KUKA KRL program: EPS_2_26115_SA7002_A_20260219035537.src

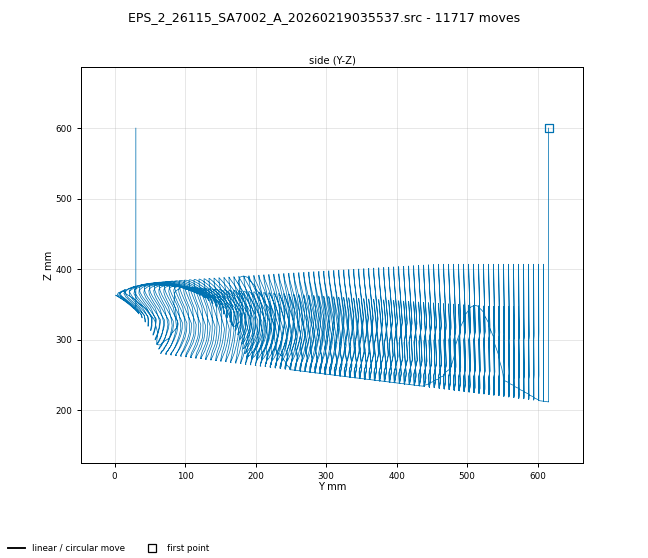
[picture p0: tool path of EPS_2_26115_SA7002_A_20260219035537.src, 11717 of 11719 moves have a stored position in this frame; points joined in program order, loops and branches not executed]
&ACCESS RVP
&REL 4
&COMMENT QRS 19112012
&PARAM EDITMASK = *
DEF PART()
EXT BAS (BAS_COMMAND :IN,REAL :IN )
INT I
BAS (#INITMOV,0 )

;KUKA QRS Post kuka4.cps  Date:22-06-2017 !

File_ID=3057

QRS_PRE_INIT()

;Init var - Until changes are made in qrs_pre_init
Outlet_Square_prg=0
Inlet_1_Square_prg=0
Inlet_2_Square_prg=0
Inlet_3_Square_prg=0
Inlet_4_Square_prg=0
Inlet_5_Square_prg=0

Outlet_1={X 0.000, Y 460.000, Z 306.500, B 0.000, E1 0.000 }
Inlet_1={X 0.000, Y 536.220, Z 246.500, B 0.000, E1 137.000 }
Outlet_1_type=201
Inlet_1_type=201
;QRS#1=Sidecore dimensions
;QRS#2=200-8" PVC SDR 35 Cut Back
;QRS#3=200-8" PVC SDR 35
;QRS#4=
;QRS#5=
;QRS#6=
;QRS#7=
;QRS#8=
;QRS#9=12-08 PSX
;QRS#10=12-08 PSX
;QRS#11=
;QRS#12=
;QRS#13=
;QRS#14=
;QRS#15=
;QRS#16=1220x127x686 2,25'
;QRS#17=EPS Height
;QRS#18=407
;QRS#19=*
;QRS#20= UPDATED VERSION 22-06-2017
;QRS#21=*
Outlet_Square=0100
Inlet_1_Square=0100
Inlet_2_Square=0
Inlet_3_Square=0
Inlet_4_Square=0
Inlet_5_Square=0
Mill_Square=1
Outlet_Square_Prg=214
Inlet_1_Square_prg=204

QRS_INIT()

$ADVANCE=5

; T1
PTP {E1 173.6,E2 173.6}
PTP {X 0,Y 615.51,A -85,B 0,C 180,E1 173.6,E2 173.6,E3 0,E4 0,E5 0,E6 0}
QRS_SPEED_INIT()
LIN {X 0,Y 615.51,Z 600,A -85,B 0,C 180,E1 173.6,E2 173.6,E3 0,E4 0,E5 0,E6 0} C_VEL
LIN {X 0,Y 615.51,Z 221.874,A -85,B 0,C 180,E1 173.6,E2 173.6} C_VEL
LIN {X 0,Y 615.51,Z 213.701,A -85,B 0,C 180,E1 173.6,E2 173.6} C_VEL
LIN {X 0,Y 615.491,Z 211.701,A -85,B 0,C 180,E1 173.414,E2 173.414} C_VEL
LIN {X 0,Y 615.474,Z 211.7,A -85,B 0,C 180,E1 170.802,E2 170.802} C_VEL
LIN {X 0,Y 615.475,Z 211.7,A -85,B 0,C 180,E1 168.808,E2 168.808} C_VEL
LIN {X 0,Y 615.494,Z 211.996,A -85,B 0,C 180,E1 168.141,E2 168.141} C_VEL
LIN {X 0,Y 615.484,Z 215.315,A -85,B 0,C 180,E1 165.452,E2 165.452} C_VEL
LIN {X 0,Y 615.469,Z 218.575,A -85,B 0,C 180,E1 162.73,E2 162.73} C_VEL
LIN {X 0,Y 615.439,Z 221.126,A -85,B 0,C 180,E1 160.662,E2 160.662} C_VEL
LIN {X 0,Y 615.437,Z 223.859,A -85,B 0,C 180,E1 158.568,E2 158.568} C_VEL
LIN {X 0,Y 615.482,Z 227.285,A -85,B 0,C 180,E1 155.991,E2 155.991} C_VEL
LIN {X 0,Y 615.455,Z 230.578,A -85,B 0,C 180,E1 153.556,E2 153.556} C_VEL
LIN {X 0,Y 615.427,Z 233.628,A -85,B 0,C 180,E1 151.341,E2 151.341} C_VEL
LIN {X 0,Y 615.423,Z 237.001,A -85,B 0,C 180,E1 148.923,E2 148.923} C_VEL
LIN {X 0,Y 615.475,Z 240.459,A -85,B 0,C 180,E1 146.467,E2 146.467} C_VEL
LIN {X 0,Y 615.481,Z 243.27,A -85,B 0,C 180,E1 144.536,E2 144.536} C_VEL
LIN {X 0,Y 615.498,Z 256.266,A -85,B 0,C 180,E1 144.248,E2 144.248} C_VEL
LIN {X 0,Y 615.471,Z 267.884,A -85,B 0,C 180,E1 143.87,E2 143.87} C_VEL
LIN {X 0,Y 615.442,Z 279.091,A -85,B 0,C 180,E1 143.384,E2 143.384} C_VEL
LIN {X 0,Y 615.469,Z 290.355,A -85,B 0,C 180,E1 142.759,E2 142.759} C_VEL
LIN {X 0,Y 615.495,Z 301.31,A -85,B 0,C 180,E1 141.986,E2 141.986} C_VEL
LIN {X 0,Y 615.498,Z 311.464,A -85,B 0,C 180,E1 141.099,E2 141.099} C_VEL
LIN {X 0,Y 615.494,Z 320.701,A -85,B 0,C 180,E1 140.081,E2 140.081} C_VEL
LIN {X 0,Y 615.496,Z 327.529,A -85,B 0,C 180,E1 139.151,E2 139.151} C_VEL
LIN {X 0,Y 615.496,Z 333.051,A -85,B 0,C 180,E1 138.224,E2 138.224} C_VEL
LIN {X 0,Y 615.495,Z 337.464,A -85,B 0,C 180,E1 137.301,E2 137.301} C_VEL
LIN {X 0,Y 615.497,Z 340.908,A -85,B 0,C 180,E1 136.381,E2 136.381} C_VEL
LIN {X 0,Y 615.498,Z 344.341,A -85,B 0,C 180,E1 135.067,E2 135.067} C_VEL
LIN {X 0,Y 615.495,Z 345.888,A -85,B 0,C 180,E1 134.001,E2 134.001} C_VEL
LIN {X 0,Y 615.496,Z 346.371,A -85,B 0,C 180,E1 133.051,E2 133.051} C_VEL
LIN {X 0,Y 615.498,Z 346.02,A -85,B 0,C 180,E1 132.084,E2 132.084} C_VEL
LIN {X 0,Y 615.495,Z 344.785,A -85,B 0,C 180,E1 131.098,E2 131.098} C_VEL
LIN {X 0,Y 615.493,Z 341.613,A -85,B 0,C 180,E1 129.749,E2 129.749} C_VEL
LIN {X 0,Y 615.492,Z 336.93,A -85,B 0,C 180,E1 128.484,E2 128.484} C_VEL
LIN {X 0,Y 615.497,Z 331.67,A -85,B 0,C 180,E1 127.434,E2 127.434} C_VEL
LIN {X 0,Y 615.496,Z 325.251,A -85,B 0,C 180,E1 126.424,E2 126.424} C_VEL
LIN {X 0,Y 615.493,Z 317.173,A -85,B 0,C 180,E1 125.414,E2 125.414} C_VEL
LIN {X 0,Y 615.497,Z 308.507,A -85,B 0,C 180,E1 124.533,E2 124.533} C_VEL
LIN {X 0,Y 615.498,Z 299.472,A -85,B 0,C 180,E1 123.78,E2 123.78} C_VEL
LIN {X 0,Y 615.481,Z 288.508,A -85,B 0,C 180,E1 123.041,E2 123.041} C_VEL
LIN {X 0,Y 615.495,Z 276.332,A -85,B 0,C 180,E1 122.395,E2 122.395} C_VEL
LIN {X 0,Y 615.48,Z 263.674,A -85,B 0,C 180,E1 121.888,E2 121.888} C_VEL
LIN {X 0,Y 615.494,Z 251.238,A -85,B 0,C 180,E1 121.535,E2 121.535} C_VEL
LIN {X 0,Y 615.485,Z 243.192,A -85,B 0,C 180,E1 121.367,E2 121.367} C_VEL
LIN {X 0,Y 615.492,Z 239.045,A -85,B 0,C 180,E1 118.455,E2 118.455} C_VEL
LIN {X 0,Y 615.476,Z 235.021,A -85,B 0,C 180,E1 115.571,E2 115.571} C_VEL
LIN {X 0,Y 615.475,Z 231.242,A -85,B 0,C 180,E1 112.844,E2 112.844} C_VEL
LIN {X 0,Y 615.485,Z 227.434,A -85,B 0,C 180,E1 110.032,E2 110.032} C_VEL
LIN {X 0,Y 615.465,Z 224.676,A -85,B 0,C 180,E1 107.957,E2 107.957} C_VEL
LIN {X 0,Y 615.45,Z 221.985,A -85,B 0,C 180,E1 105.906,E2 105.906} C_VEL
LIN {X 0,Y 615.439,Z 219.39,A -85,B 0,C 180,E1 103.875,E2 103.875} C_VEL
LIN {X 0,Y 615.481,Z 216.126,A -85,B 0,C 180,E1 101.193,E2 101.193} C_VEL
LIN {X 0,Y 615.476,Z 212.873,A -85,B 0,C 180,E1 98.536,E2 98.536} C_VEL
LIN {X 0,Y 615.485,Z 212.061,A -85,B 0,C 180,E1 97.875,E2 97.875} C_VEL
LIN {X 0,Y 615.497,Z 211.7,A -85,B 0,C 180,E1 96.556,E2 96.556} C_VEL
LIN {X 0,Y 615.482,Z 211.7,A -85,B 0,C 180,E1 93.928,E2 93.928} C_VEL
LIN {X 0,Y 615.487,Z 211.696,A -85,B 0,C 180,E1 91.308,E2 91.308} C_VEL
LIN {X 0,Y 615.484,Z 211.696,A -85,B 0,C 180,E1 88.691,E2 88.691} C_VEL
LIN {X 0,Y 615.476,Z 211.7,A -85,B 0,C 180,E1 86.071,E2 86.071} C_VEL
LIN {X 0,Y 615.491,Z 211.702,A -85,B 0,C 180,E1 83.402,E2 83.402} C_VEL
LIN {X 0,Y 615.475,Z 211.701,A -85,B 0,C 180,E1 80.801,E2 80.801} C_VEL
LIN {X 0,Y 615.468,Z 211.7,A -85,B 0,C 180,E1 78.139,E2 78.139} C_VEL
LIN {X 0,Y 615.482,Z 211.697,A -85,B 0,C 180,E1 75.451,E2 75.451} C_VEL
LIN {X 0,Y 615.497,Z 211.699,A -85,B 0,C 180,E1 72.729,E2 72.729} C_VEL
LIN {X 0,Y 615.481,Z 211.698,A -85,B 0,C 180,E1 69.967,E2 69.967} C_VEL
LIN {X 0,Y 615.49,Z 211.695,A -85,B 0,C 180,E1 67.155,E2 67.155} C_VEL
LIN {X 0,Y 615.496,Z 211.7,A -85,B 0,C 180,E1 64.284,E2 64.284} C_VEL
LIN {X 0,Y 615.489,Z 211.695,A -85,B 0,C 180,E1 61.342,E2 61.342} C_VEL
LIN {X 0,Y 615.47,Z 211.699,A -85,B 0,C 180,E1 58.913,E2 58.913} C_VEL
LIN {X 0,Y 615.466,Z 211.7,A -85,B 0,C 180,E1 56.466,E2 56.466} C_VEL
LIN {X 0,Y 615.465,Z 211.7,A -85,B 0,C 180,E1 54.166,E2 54.166} C_VEL
LIN {X 0,Y 615.487,Z 211.696,A -85,B 0,C 180,E1 51.931,E2 51.931} C_VEL
LIN {X 0,Y 615.486,Z 211.696,A -85,B 0,C 180,E1 49.393,E2 49.393} C_VEL
LIN {X 0,Y 615.475,Z 211.7,A -85,B 0,C 180,E1 46.754,E2 46.754} C_VEL
LIN {X 0,Y 615.495,Z 211.699,A -85,B 0,C 180,E1 43.998,E2 43.998} C_VEL
LIN {X 0,Y 615.466,Z 211.7,A -85,B 0,C 180,E1 41.092,E2 41.092} C_VEL
LIN {X 0,Y 615.468,Z 211.701,A -85,B 0,C 180,E1 38.904,E2 38.904} C_VEL
LIN {X 0,Y 615.476,Z 211.698,A -85,B 0,C 180,E1 36.424,E2 36.424} C_VEL
LIN {X 0,Y 615.493,Z 211.698,A -85,B 0,C 180,E1 33.535,E2 33.535} C_VEL
LIN {X 0,Y 615.488,Z 211.702,A -85,B 0,C 180,E1 30.918,E2 30.918} C_VEL
LIN {X 0,Y 615.492,Z 211.699,A -85,B 0,C 180,E1 28.451,E2 28.451} C_VEL
LIN {X 0,Y 615.474,Z 211.698,A -85,B 0,C 180,E1 25.566,E2 25.566} C_VEL
LIN {X 0,Y 615.478,Z 211.701,A -85,B 0,C 180,E1 22.843,E2 22.843} C_VEL
LIN {X 0,Y 615.474,Z 211.7,A -85,B 0,C 180,E1 20.553,E2 20.553} C_VEL
LIN {X 0,Y 615.497,Z 211.698,A -85,B 0,C 180,E1 17.955,E2 17.955} C_VEL
LIN {X 0,Y 615.478,Z 211.7,A -85,B 0,C 180,E1 15.225,E2 15.225} C_VEL
LIN {X 0,Y 615.488,Z 211.695,A -85,B 0,C 180,E1 12.529,E2 12.529} C_VEL
LIN {X 0,Y 615.483,Z 211.698,A -85,B 0,C 180,E1 9.861,E2 9.861} C_VEL
LIN {X 0,Y 615.486,Z 211.701,A -85,B 0,C 180,E1 7.214,E2 7.214} C_VEL
LIN {X 0,Y 615.496,Z 211.697,A -85,B 0,C 180,E1 4.583,E2 4.583} C_VEL
LIN {X 0,Y 615.471,Z 211.7,A -85,B 0,C 180,E1 1.962,E2 1.962} C_VEL
LIN {X 0,Y 615.467,Z 211.7,A -85,B 0,C 180,E1 -0.655,E2 -0.655} C_VEL
LIN {X 0,Y 615.484,Z 211.698,A -85,B 0,C 180,E1 -3.274,E2 -3.274} C_VEL
LIN {X 0,Y 615.495,Z 211.699,A -85,B 0,C 180,E1 -5.899,E2 -5.899} C_VEL
LIN {X 0,Y 615.485,Z 211.7,A -85,B 0,C 180,E1 -8.538,E2 -8.538} C_VEL
LIN {X 0,Y 615.49,Z 211.695,A -85,B 0,C 180,E1 -11.194,E2 -11.194} C_VEL
LIN {X 0,Y 615.475,Z 211.699,A -85,B 0,C 180,E1 -13.927,E2 -13.927} C_VEL
LIN {X 0,Y 615.488,Z 211.7,A -85,B 0,C 180,E1 -16.587,E2 -16.587} C_VEL
LIN {X 0,Y 615.486,Z 211.698,A -85,B 0,C 180,E1 -19.339,E2 -19.339} C_VEL
LIN {X 0,Y 615.466,Z 211.7,A -85,B 0,C 180,E1 -22.138,E2 -22.138} C_VEL
LIN {X 0,Y 615.493,Z 211.7,A -85,B 0,C 180,E1 -24.992,E2 -24.992} C_VEL
LIN {X 0,Y 615.497,Z 211.696,A -85,B 0,C 180,E1 -27.178,E2 -27.178} C_VEL
LIN {X 0,Y 615.499,Z 211.7,A -85,B 0,C 180,E1 -29.796,E2 -29.796} C_VEL
LIN {X 0,Y 615.488,Z 211.698,A -85,B 0,C 180,E1 -32.458,E2 -32.458} C_VEL
LIN {X 0,Y 615.497,Z 211.696,A -85,B 0,C 180,E1 -34.815,E2 -34.815} C_VEL
LIN {X 0,Y 615.476,Z 211.7,A -85,B 0,C 180,E1 -37.244,E2 -37.244} C_VEL
LIN {X 0,Y 615.469,Z 211.7,A -85,B 0,C 180,E1 -39.752,E2 -39.752} C_VEL
LIN {X 0,Y 615.473,Z 211.699,A -85,B 0,C 180,E1 -42.355,E2 -42.355} C_VEL
LIN {X 0,Y 615.49,Z 211.698,A -85,B 0,C 180,E1 -45.069,E2 -45.069} C_VEL
LIN {X 0,Y 615.484,Z 211.699,A -85,B 0,C 180,E1 -47.921,E2 -47.921} C_VEL
LIN {X 0,Y 615.491,Z 211.696,A -85,B 0,C 180,E1 -50.938,E2 -50.938} C_VEL
LIN {X 0,Y 615.486,Z 211.701,A -85,B 0,C 180,E1 -53.575,E2 -53.575} C_VEL
LIN {X 0,Y 615.49,Z 211.816,A -85,B 0,C 180,E1 -54.535,E2 -54.535} C_VEL
LIN {X 0,Y 615.437,Z 220.579,A -85,B 0,C 180,E1 -57.151,E2 -57.151} C_VEL
LIN {X 0,Y 615.425,Z 228.512,A -85,B 0,C 180,E1 -59.457,E2 -59.457} C_VEL
LIN {X 0,Y 615.48,Z 237.754,A -85,B 0,C 180,E1 -62.084,E2 -62.084} C_VEL
LIN {X 0,Y 615.47,Z 247.263,A -85,B 0,C 180,E1 -64.718,E2 -64.718} C_VEL
LIN {X 0,Y 615.465,Z 256.236,A -85,B 0,C 180,E1 -67.154,E2 -67.154} C_VEL
LIN {X 0,Y 615.483,Z 266.781,A -85,B 0,C 180,E1 -69.967,E2 -69.967} C_VEL
LIN {X 0,Y 615.484,Z 277.325,A -85,B 0,C 180,E1 -72.729,E2 -72.729} C_VEL
LIN {X 0,Y 615.464,Z 287.861,A -85,B 0,C 180,E1 -75.45,E2 -75.45} C_VEL
LIN {X 0,Y 615.484,Z 298.39,A -85,B 0,C 180,E1 -78.139,E2 -78.139} C_VEL
LIN {X 0,Y 615.496,Z 299.207,A -85,B 0,C 180,E1 -78.348,E2 -78.348} C_VEL
LIN {X 0,Y 615.497,Z 313.809,A -85,B 0,C 180,E1 -78.64,E2 -78.64} C_VEL
LIN {X 0,Y 615.455,Z 326.946,A -85,B 0,C 180,E1 -79.05,E2 -79.05} C_VEL
LIN {X 0,Y 615.447,Z 338.766,A -85,B 0,C 180,E1 -79.555,E2 -79.555} C_VEL
LIN {X 0,Y 615.497,Z 349.381,A -85,B 0,C 180,E1 -80.138,E2 -80.138} C_VEL
LIN {X 0,Y 615.498,Z 360.228,A -85,B 0,C 180,E1 -80.884,E2 -80.884} C_VEL
LIN {X 0,Y 615.497,Z 370.808,A -85,B 0,C 180,E1 -81.794,E2 -81.794} C_VEL
LIN {X 0,Y 615.498,Z 378.603,A -85,B 0,C 180,E1 -82.619,E2 -82.619} C_VEL
LIN {X 0,Y 615.496,Z 386.201,A -85,B 0,C 180,E1 -83.608,E2 -83.608} C_VEL
LIN {X 0,Y 615.498,Z 393.203,A -85,B 0,C 180,E1 -84.759,E2 -84.759} C_VEL
LIN {X 0,Y 615.494,Z 397.85,A -85,B 0,C 180,E1 -85.743,E2 -85.743} C_VEL
LIN {X 0,Y 615.494,Z 401.398,A -85,B 0,C 180,E1 -86.727,E2 -86.727} C_VEL
LIN {X 0,Y 615.497,Z 403.232,A -85,B 0,C 180,E1 -87.382,E2 -87.382} C_VEL
LIN {X 0,Y 615.5,Z 404.607,A -85,B 0,C 180,E1 -88.037,E2 -88.037} C_VEL
LIN {X 0,Y 615.496,Z 406.173,A -85,B 0,C 180,E1 -89.345,E2 -89.345} C_VEL
LIN {X 0,Y 615.494,Z 406.389,A -85,B 0,C 180,E1 -90,E2 -90} C_VEL
LIN {X 0,Y 615.495,Z 405.58,A -85,B 0,C 180,E1 -91.308,E2 -91.308} C_VEL
LIN {X 0,Y 615.5,Z 404.608,A -85,B 0,C 180,E1 -91.963,E2 -91.963} C_VEL
LIN {X 0,Y 615.497,Z 403.234,A -85,B 0,C 180,E1 -92.617,E2 -92.617} C_VEL
LIN {X 0,Y 615.496,Z 400.351,A -85,B 0,C 180,E1 -93.6,E2 -93.6} C_VEL
LIN {X 0,Y 615.498,Z 396.443,A -85,B 0,C 180,E1 -94.584,E2 -94.584} C_VEL
LIN {X 0,Y 615.499,Z 391.407,A -85,B 0,C 180,E1 -95.569,E2 -95.569} C_VEL
LIN {X 0,Y 615.497,Z 384.871,A -85,B 0,C 180,E1 -96.583,E2 -96.583} C_VEL
LIN {X 0,Y 615.497,Z 377.137,A -85,B 0,C 180,E1 -97.545,E2 -97.545} C_VEL
LIN {X 0,Y 615.498,Z 369.049,A -85,B 0,C 180,E1 -98.371,E2 -98.371} C_VEL
LIN {X 0,Y 615.499,Z 359.173,A -85,B 0,C 180,E1 -99.198,E2 -99.198} C_VEL
LIN {X 0,Y 615.486,Z 347.989,A -85,B 0,C 180,E1 -99.945,E2 -99.945} C_VEL
LIN {X 0,Y 615.445,Z 337.038,A -85,B 0,C 180,E1 -100.527,E2 -100.527} C_VEL
LIN {X 0,Y 615.461,Z 324.766,A -85,B 0,C 180,E1 -101.031,E2 -101.031} C_VEL
LIN {X 0,Y 615.499,Z 312.081,A -85,B 0,C 180,E1 -101.401,E2 -101.401} C_VEL
LIN {X 0,Y 615.496,Z 299.21,A -85,B 0,C 180,E1 -101.651,E2 -101.651} C_VEL
LIN {X 0,Y 615.465,Z 289.075,A -85,B 0,C 180,E1 -104.24,E2 -104.24} C_VEL
LIN {X 0,Y 615.49,Z 278.641,A -85,B 0,C 180,E1 -106.928,E2 -106.928} C_VEL
LIN {X 0,Y 615.487,Z 268.106,A -85,B 0,C 180,E1 -109.685,E2 -109.685} C_VEL
LIN {X 0,Y 615.491,Z 258.087,A -85,B 0,C 180,E1 -112.346,E2 -112.346} C_VEL
LIN {X 0,Y 615.456,Z 248.325,A -85,B 0,C 180,E1 -114.993,E2 -114.993} C_VEL
LIN {X 0,Y 615.494,Z 239.076,A -85,B 0,C 180,E1 -117.545,E2 -117.545} C_VEL
LIN {X 0,Y 615.44,Z 229.836,A -85,B 0,C 180,E1 -120.162,E2 -120.162} C_VEL
LIN {X 0,Y 615.421,Z 221.905,A -85,B 0,C 180,E1 -122.461,E2 -122.461} C_VEL
LIN {X 0,Y 615.454,Z 213.969,A -85,B 0,C 180,E1 -124.817,E2 -124.817} C_VEL
LIN {X 0,Y 615.492,Z 211.697,A -85,B 0,C 180,E1 -125.514,E2 -125.514} C_VEL
LIN {X 0,Y 615.486,Z 211.699,A -85,B 0,C 180,E1 -128.068,E2 -128.068} C_VEL
LIN {X 0,Y 615.484,Z 211.7,A -85,B 0,C 180,E1 -130.606,E2 -130.606} C_VEL
LIN {X 0,Y 615.497,Z 211.697,A -85,B 0,C 180,E1 -133.243,E2 -133.243} C_VEL
LIN {X 0,Y 615.474,Z 211.7,A -85,B 0,C 180,E1 -136.003,E2 -136.003} C_VEL
LIN {X 0,Y 615.487,Z 211.7,A -85,B 0,C 180,E1 -138.525,E2 -138.525} C_VEL
LIN {X 0,Y 615.495,Z 211.696,A -85,B 0,C 180,E1 -141.096,E2 -141.096} C_VEL
LIN {X 0,Y 615.487,Z 211.698,A -85,B 0,C 180,E1 -143.574,E2 -143.574} C_VEL
LIN {X 0,Y 615.495,Z 211.701,A -85,B 0,C 180,E1 -145.978,E2 -145.978} C_VEL
LIN {X 0,Y 615.484,Z 211.7,A -85,B 0,C 180,E1 -148.913,E2 -148.913} C_VEL
LIN {X 0,Y 615.475,Z 211.7,A -85,B 0,C 180,E1 -151.551,E2 -151.551} C_VEL
LIN {X 0,Y 615.498,Z 211.7,A -85,B 0,C 180,E1 -154.284,E2 -154.284} C_VEL
LIN {X 0,Y 615.493,Z 211.697,A -85,B 0,C 180,E1 -157.155,E2 -157.155} C_VEL
LIN {X 0,Y 615.475,Z 211.7,A -85,B 0,C 180,E1 -159.966,E2 -159.966} C_VEL
LIN {X 0,Y 615.497,Z 211.699,A -85,B 0,C 180,E1 -162.729,E2 -162.729} C_VEL
LIN {X 0,Y 615.481,Z 211.7,A -85,B 0,C 180,E1 -165.45,E2 -165.45} C_VEL
LIN {X 0,Y 615.484,Z 211.699,A -85,B 0,C 180,E1 -168.138,E2 -168.138} C_VEL
LIN {X 0,Y 615.496,Z 211.698,A -85,B 0,C 180,E1 -170.8,E2 -170.8} C_VEL
LIN {X 0,Y 615.474,Z 211.7,A -85,B 0,C 180,E1 -173.442,E2 -173.442} C_VEL
LIN {X 0,Y 615.488,Z 211.701,A -85,B 0,C 180,E1 -176.07,E2 -176.07} C_VEL
LIN {X 0,Y 615.491,Z 211.696,A -85,B 0,C 180,E1 -178.69,E2 -178.69} C_VEL
LIN {X 0,Y 615.496,Z 211.7,A -85,B 0,C 180,E1 -181.307,E2 -181.307} C_VEL
LIN {X 0,Y 615.477,Z 211.7,A -85,B 0,C 180,E1 -183.927,E2 -183.927} C_VEL
LIN {X 0,Y 615.491,Z 211.701,A -85,B 0,C 180,E1 -186.586,E2 -186.586} C_VEL
LIN {X 0,Y 614.803,Z 211.847,A -85,B 0,C 180,E1 -187.132,E2 -187.132} C_VEL
LIN {X 0,Y 611.958,Z 212.259,A -85,B 0,C 180,E1 -188.018,E2 -188.018} C_VEL
LIN {X 0,Y 609.568,Z 212.568,A -85,B 0,C 180,E1 -188.731,E2 -188.731} C_VEL
LIN {X 0,Y 608.539,Z 212.686,A -85,B 0,C 180,E1 -189.28,E2 -189.28} C_VEL
LIN {X 0,Y 608.454,Z 212.695,A -85,B 0,C 180,E1 -189.466,E2 -189.466} C_VEL
LIN {X 0,Y 608.44,Z 212.697,A -85,B 0,C 180,E1 -191.323,E2 -191.323} C_VEL
LIN {X 0,Y 608.449,Z 213.027,A -85,B 0,C 180,E1 -191.999,E2 -191.999} C_VEL
LIN {X 0,Y 608.442,Z 216.384,A -85,B 0,C 180,E1 -194.72,E2 -194.72} C_VEL
LIN {X 0,Y 608.437,Z 219.656,A -85,B 0,C 180,E1 -197.476,E2 -197.476} C_VEL
LIN {X 0,Y 608.426,Z 223.103,A -85,B 0,C 180,E1 -200.274,E2 -200.274} C_VEL
LIN {X 0,Y 608.374,Z 226.848,A -85,B 0,C 180,E1 -203.125,E2 -203.125} C_VEL
LIN {X 0,Y 608.389,Z 230.305,A -85,B 0,C 180,E1 -205.706,E2 -205.706} C_VEL
LIN {X 0,Y 608.366,Z 234.261,A -85,B 0,C 180,E1 -208.603,E2 -208.603} C_VEL
LIN {X 0,Y 608.396,Z 236.953,A -85,B 0,C 180,E1 -210.547,E2 -210.547} C_VEL
LIN {X 0,Y 608.388,Z 240.222,A -85,B 0,C 180,E1 -212.882,E2 -212.882} C_VEL
LIN {X 0,Y 608.407,Z 243.684,A -85,B 0,C 180,E1 -215.329,E2 -215.329} C_VEL
LIN {X 0,Y 608.536,Z 257.877,A -85,B 0,C 180,E1 -215.663,E2 -215.663} C_VEL
LIN {X 0,Y 608.509,Z 270.159,A -85,B 0,C 180,E1 -216.086,E2 -216.086} C_VEL
LIN {X 0,Y 608.464,Z 281.367,A -85,B 0,C 180,E1 -216.603,E2 -216.603} C_VEL
LIN {X 0,Y 608.475,Z 292.485,A -85,B 0,C 180,E1 -217.255,E2 -217.255} C_VEL
LIN {X 0,Y 608.483,Z 302.616,A -85,B 0,C 180,E1 -217.993,E2 -217.993} C_VEL
LIN {X 0,Y 608.459,Z 311.688,A -85,B 0,C 180,E1 -218.799,E2 -218.799} C_VEL
LIN {X 0,Y 608.467,Z 319.57,A -85,B 0,C 180,E1 -219.652,E2 -219.652} C_VEL
LIN {X 0,Y 608.451,Z 327.678,A -85,B 0,C 180,E1 -220.736,E2 -220.736} C_VEL
LIN {X 0,Y 608.444,Z 334.345,A -85,B 0,C 180,E1 -221.867,E2 -221.867} C_VEL
LIN {X 0,Y 608.436,Z 339.259,A -85,B 0,C 180,E1 -222.959,E2 -222.959} C_VEL
LIN {X 0,Y 608.423,Z 343.45,A -85,B 0,C 180,E1 -224.261,E2 -224.261} C_VEL
LIN {X 0,Y 608.419,Z 345.438,A -85,B 0,C 180,E1 -225.201,E2 -225.201} C_VEL
LIN {X 0,Y 608.427,Z 346.604,A -85,B 0,C 180,E1 -226.128,E2 -226.128} C_VEL
LIN {X 0,Y 608.434,Z 347,A -85,B 0,C 180,E1 -227.039,E2 -227.039} C_VEL
LIN {X 0,Y 608.425,Z 346.622,A -85,B 0,C 180,E1 -227.936,E2 -227.936} C_VEL
LIN {X 0,Y 608.43,Z 345.548,A -85,B 0,C 180,E1 -228.822,E2 -228.822} C_VEL
LIN {X 0,Y 608.436,Z 342.648,A -85,B 0,C 180,E1 -230.129,E2 -230.129} C_VEL
LIN {X 0,Y 608.435,Z 339.537,A -85,B 0,C 180,E1 -231.057,E2 -231.057} C_VEL
LIN {X 0,Y 608.437,Z 334.197,A -85,B 0,C 180,E1 -232.252,E2 -232.252} C_VEL
LIN {X 0,Y 608.448,Z 328.095,A -85,B 0,C 180,E1 -233.292,E2 -233.292} C_VEL
LIN {X 0,Y 608.448,Z 320.381,A -85,B 0,C 180,E1 -234.339,E2 -234.339} C_VEL
LIN {X 0,Y 608.481,Z 311.467,A -85,B 0,C 180,E1 -235.313,E2 -235.313} C_VEL
LIN {X 0,Y 608.474,Z 302.254,A -85,B 0,C 180,E1 -236.126,E2 -236.126} C_VEL
LIN {X 0,Y 608.484,Z 291.108,A -85,B 0,C 180,E1 -236.925,E2 -236.925} C_VEL
LIN {X 0,Y 608.498,Z 279.579,A -85,B 0,C 180,E1 -237.578,E2 -237.578} C_VEL
LIN {X 0,Y 608.515,Z 267.528,A -85,B 0,C 180,E1 -238.104,E2 -238.104} C_VEL
LIN {X 0,Y 608.553,Z 254.097,A -85,B 0,C 180,E1 -238.532,E2 -238.532} C_VEL
LIN {X 0,Y 608.413,Z 243.683,A -85,B 0,C 180,E1 -238.762,E2 -238.762} C_VEL
LIN {X 0,Y 608.416,Z 239.971,A -85,B 0,C 180,E1 -241.386,E2 -241.386} C_VEL
LIN {X 0,Y 608.423,Z 235.921,A -85,B 0,C 180,E1 -244.284,E2 -244.284} C_VEL
LIN {X 0,Y 608.409,Z 232.355,A -85,B 0,C 180,E1 -246.875,E2 -246.875} C_VEL
LIN {X 0,Y 608.428,Z 228.498,A -85,B 0,C 180,E1 -249.725,E2 -249.725} C_VEL
LIN {X 0,Y 608.402,Z 224.791,A -85,B 0,C 180,E1 -252.522,E2 -252.522} C_VEL
LIN {X 0,Y 608.438,Z 221.239,A -85,B 0,C 180,E1 -255.279,E2 -255.279} C_VEL
LIN {X 0,Y 608.381,Z 217.947,A -85,B 0,C 180,E1 -257.999,E2 -257.999} C_VEL
LIN {X 0,Y 608.431,Z 215.482,A -85,B 0,C 180,E1 -260.023,E2 -260.023} C_VEL
LIN {X 0,Y 608.44,Z 213.023,A -85,B 0,C 180,E1 -262.033,E2 -262.033} C_VEL
LIN {X 0,Y 608.479,Z 212.694,A -85,B 0,C 180,E1 -263.368,E2 -263.368} C_VEL
LIN {X 0,Y 608.451,Z 212.697,A -85,B 0,C 180,E1 -266.026,E2 -266.026} C_VEL
LIN {X 0,Y 608.469,Z 212.693,A -85,B 0,C 180,E1 -268.677,E2 -268.677} C_VEL
LIN {X 0,Y 608.467,Z 212.693,A -85,B 0,C 180,E1 -271.324,E2 -271.324} C_VEL
LIN {X 0,Y 608.445,Z 212.697,A -85,B 0,C 180,E1 -273.974,E2 -273.974} C_VEL
LIN {X 0,Y 608.46,Z 212.697,A -85,B 0,C 180,E1 -276.633,E2 -276.633} C_VEL
LIN {X 0,Y 608.458,Z 212.695,A -85,B 0,C 180,E1 -279.306,E2 -279.306} C_VEL
LIN {X 0,Y 608.448,Z 212.695,A -85,B 0,C 180,E1 -282,E2 -282} C_VEL
LIN {X 0,Y 608.468,Z 212.694,A -85,B 0,C 180,E1 -284.721,E2 -284.721} C_VEL
LIN {X 0,Y 608.452,Z 212.697,A -85,B 0,C 180,E1 -287.477,E2 -287.477} C_VEL
LIN {X 0,Y 608.46,Z 212.693,A -85,B 0,C 180,E1 -290.275,E2 -290.275} C_VEL
LIN {X 0,Y 608.448,Z 212.697,A -85,B 0,C 180,E1 -293.124,E2 -293.124} C_VEL
LIN {X 0,Y 608.452,Z 212.695,A -85,B 0,C 180,E1 -296.036,E2 -296.036} C_VEL
LIN {X 0,Y 608.476,Z 212.691,A -85,B 0,C 180,E1 -298.624,E2 -298.624} C_VEL
LIN {X 0,Y 608.465,Z 212.694,A -85,B 0,C 180,E1 -301.317,E2 -301.317} C_VEL
LIN {X 0,Y 608.462,Z 212.694,A -85,B 0,C 180,E1 -303.737,E2 -303.737} C_VEL
LIN {X 0,Y 608.448,Z 212.696,A -85,B 0,C 180,E1 -306.092,E2 -306.092} C_VEL
LIN {X 0,Y 608.467,Z 212.695,A -85,B 0,C 180,E1 -308.588,E2 -308.588} C_VEL
LIN {X 0,Y 608.456,Z 212.696,A -85,B 0,C 180,E1 -311.344,E2 -311.344} C_VEL
LIN {X 0,Y 608.46,Z 212.694,A -85,B 0,C 180,E1 -314.267,E2 -314.267} C_VEL
LIN {X 0,Y 608.453,Z 212.697,A -85,B 0,C 180,E1 -317.043,E2 -317.043} C_VEL
LIN {X 0,Y 608.455,Z 212.696,A -85,B 0,C 180,E1 -319.699,E2 -319.699} C_VEL
LIN {X 0,Y 608.47,Z 212.693,A -85,B 0,C 180,E1 -322.256,E2 -322.256} C_VEL
LIN {X 0,Y 608.44,Z 212.696,A -85,B 0,C 180,E1 -324.724,E2 -324.724} C_VEL
LIN {X 0,Y 608.454,Z 212.694,A -85,B 0,C 180,E1 -327.122,E2 -327.122} C_VEL
LIN {X 0,Y 608.472,Z 212.692,A -85,B 0,C 180,E1 -329.457,E2 -329.457} C_VEL
LIN {X 0,Y 608.457,Z 212.695,A -85,B 0,C 180,E1 -331.735,E2 -331.735} C_VEL
LIN {X 0,Y 608.462,Z 212.693,A -85,B 0,C 180,E1 -334.281,E2 -334.281} C_VEL
LIN {X 0,Y 608.443,Z 212.696,A -85,B 0,C 180,E1 -336.877,E2 -336.877} C_VEL
LIN {X 0,Y 608.456,Z 212.694,A -85,B 0,C 180,E1 -339.325,E2 -339.325} C_VEL
LIN {X 0,Y 608.455,Z 212.695,A -85,B 0,C 180,E1 -341.83,E2 -341.83} C_VEL
LIN {X 0,Y 608.466,Z 212.696,A -85,B 0,C 180,E1 -344.595,E2 -344.595} C_VEL
LIN {X 0,Y 608.477,Z 212.692,A -85,B 0,C 180,E1 -347.324,E2 -347.324} C_VEL
LIN {X 0,Y 608.455,Z 212.694,A -85,B 0,C 180,E1 -350.024,E2 -350.024} C_VEL
LIN {X 0,Y 608.463,Z 212.695,A -85,B 0,C 180,E1 -352.702,E2 -352.702} C_VEL
LIN {X 0,Y 608.462,Z 212.696,A -85,B 0,C 180,E1 -355.364,E2 -355.364} C_VEL
LIN {X 0,Y 608.441,Z 212.696,A -85,B 0,C 180,E1 -358.015,E2 -358.015} C_VEL
LIN {X 0,Y 608.464,Z 212.693,A -85,B 0,C 180,E1 -360.663,E2 -360.663} C_VEL
LIN {X 0,Y 608.477,Z 212.692,A -85,B 0,C 180,E1 -363.312,E2 -363.312} C_VEL
LIN {X 0,Y 608.466,Z 212.697,A -85,B 0,C 180,E1 -365.968,E2 -365.968} C_VEL
LIN {X 0,Y 608.456,Z 212.695,A -85,B 0,C 180,E1 -368.637,E2 -368.637} C_VEL
LIN {X 0,Y 608.481,Z 212.691,A -85,B 0,C 180,E1 -371.325,E2 -371.325} C_VEL
LIN {X 0,Y 608.451,Z 212.696,A -85,B 0,C 180,E1 -374.039,E2 -374.039} C_VEL
LIN {X 0,Y 608.48,Z 212.694,A -85,B 0,C 180,E1 -376.784,E2 -376.784} C_VEL
LIN {X 0,Y 608.451,Z 212.695,A -85,B 0,C 180,E1 -379.571,E2 -379.571} C_VEL
LIN {X 0,Y 608.464,Z 212.695,A -85,B 0,C 180,E1 -382.477,E2 -382.477} C_VEL
LIN {X 0,Y 608.443,Z 212.697,A -85,B 0,C 180,E1 -385.302,E2 -385.302} C_VEL
LIN {X 0,Y 608.448,Z 212.698,A -85,B 0,C 180,E1 -387.519,E2 -387.519} C_VEL
LIN {X 0,Y 608.454,Z 212.696,A -85,B 0,C 180,E1 -389.969,E2 -389.969} C_VEL
LIN {X 0,Y 608.464,Z 212.693,A -85,B 0,C 180,E1 -392.88,E2 -392.88} C_VEL
LIN {X 0,Y 608.449,Z 212.695,A -85,B 0,C 180,E1 -395.278,E2 -395.278} C_VEL
LIN {X 0,Y 608.473,Z 212.695,A -85,B 0,C 180,E1 -398.241,E2 -398.241} C_VEL
LIN {X 0,Y 608.461,Z 212.694,A -85,B 0,C 180,E1 -401.342,E2 -401.342} C_VEL
LIN {X 0,Y 608.465,Z 212.695,A -85,B 0,C 180,E1 -404.265,E2 -404.265} C_VEL
LIN {X 0,Y 608.452,Z 212.694,A -85,B 0,C 180,E1 -407.04,E2 -407.04} C_VEL
LIN {X 0,Y 608.458,Z 212.694,A -85,B 0,C 180,E1 -409.697,E2 -409.697} C_VEL
LIN {X 0,Y 608.459,Z 212.695,A -85,B 0,C 180,E1 -412.253,E2 -412.253} C_VEL
LIN {X 0,Y 608.483,Z 212.814,A -85,B 0,C 180,E1 -414.369,E2 -414.369} C_VEL
LIN {X 0,Y 608.491,Z 221.916,A -85,B 0,C 180,E1 -417.122,E2 -417.122} C_VEL
LIN {X 0,Y 608.456,Z 229.859,A -85,B 0,C 180,E1 -419.454,E2 -419.454} C_VEL
LIN {X 0,Y 608.494,Z 239.126,A -85,B 0,C 180,E1 -422.11,E2 -422.11} C_VEL
LIN {X 0,Y 608.461,Z 248.394,A -85,B 0,C 180,E1 -424.699,E2 -424.699} C_VEL
LIN {X 0,Y 608.448,Z 257.662,A -85,B 0,C 180,E1 -427.235,E2 -427.235} C_VEL
LIN {X 0,Y 608.463,Z 266.928,A -85,B 0,C 180,E1 -429.726,E2 -429.726} C_VEL
LIN {X 0,Y 608.463,Z 277.519,A -85,B 0,C 180,E1 -432.523,E2 -432.523} C_VEL
LIN {X 0,Y 608.437,Z 288.11,A -85,B 0,C 180,E1 -435.278,E2 -435.278} C_VEL
LIN {X 0,Y 608.423,Z 297.378,A -85,B 0,C 180,E1 -437.661,E2 -437.661} C_VEL
LIN {X 0,Y 608.443,Z 299.529,A -85,B 0,C 180,E1 -438.211,E2 -438.211} C_VEL
LIN {X 0,Y 608.546,Z 314.685,A -85,B 0,C 180,E1 -438.53,E2 -438.53} C_VEL
LIN {X 0,Y 608.478,Z 327.499,A -85,B 0,C 180,E1 -438.939,E2 -438.939} C_VEL
LIN {X 0,Y 608.474,Z 338.914,A -85,B 0,C 180,E1 -439.434,E2 -439.434} C_VEL
LIN {X 0,Y 608.486,Z 349.573,A -85,B 0,C 180,E1 -440.023,E2 -440.023} C_VEL
LIN {X 0,Y 608.483,Z 360.47,A -85,B 0,C 180,E1 -440.778,E2 -440.778} C_VEL
LIN {X 0,Y 608.475,Z 371.108,A -85,B 0,C 180,E1 -441.698,E2 -441.698} C_VEL
LIN {X 0,Y 608.471,Z 378.957,A -85,B 0,C 180,E1 -442.534,E2 -442.534} C_VEL
LIN {X 0,Y 608.461,Z 386.286,A -85,B 0,C 180,E1 -443.484,E2 -443.484} C_VEL
LIN {X 0,Y 608.451,Z 391.864,A -85,B 0,C 180,E1 -444.365,E2 -444.365} C_VEL
LIN {X 0,Y 608.432,Z 396.949,A -85,B 0,C 180,E1 -445.362,E2 -445.362} C_VEL
LIN {X 0,Y 608.449,Z 400.895,A -85,B 0,C 180,E1 -446.357,E2 -446.357} C_VEL
LIN {X 0,Y 608.425,Z 403.808,A -85,B 0,C 180,E1 -447.351,E2 -447.351} C_VEL
LIN {X 0,Y 608.445,Z 405.201,A -85,B 0,C 180,E1 -448.014,E2 -448.014} C_VEL
LIN {X 0,Y 608.439,Z 406.783,A -85,B 0,C 180,E1 -449.338,E2 -449.338} C_VEL
LIN {X 0,Y 608.434,Z 407,A -85,B 0,C 180,E1 -450,E2 -450} C_VEL
LIN {X 0,Y 608.448,Z 406.184,A -85,B 0,C 180,E1 -451.323,E2 -451.323} C_VEL
LIN {X 0,Y 608.444,Z 405.202,A -85,B 0,C 180,E1 -451.985,E2 -451.985} C_VEL
LIN {X 0,Y 608.425,Z 403.81,A -85,B 0,C 180,E1 -452.648,E2 -452.648} C_VEL
LIN {X 0,Y 608.449,Z 400.897,A -85,B 0,C 180,E1 -453.642,E2 -453.642} C_VEL
LIN {X 0,Y 608.432,Z 396.952,A -85,B 0,C 180,E1 -454.637,E2 -454.637} C_VEL
LIN {X 0,Y 608.438,Z 390.879,A -85,B 0,C 180,E1 -455.8,E2 -455.8} C_VEL
LIN {X 0,Y 608.462,Z 384.238,A -85,B 0,C 180,E1 -456.799,E2 -456.799} C_VEL
LIN {X 0,Y 608.456,Z 375.993,A -85,B 0,C 180,E1 -457.8,E2 -457.8} C_VEL
LIN {X 0,Y 608.472,Z 367.541,A -85,B 0,C 180,E1 -458.635,E2 -458.635} C_VEL
LIN {X 0,Y 608.481,Z 357.096,A -85,B 0,C 180,E1 -459.473,E2 -459.473} C_VEL
LIN {X 0,Y 608.494,Z 346.762,A -85,B 0,C 180,E1 -460.144,E2 -460.144} C_VEL
LIN {X 0,Y 608.469,Z 335.847,A -85,B 0,C 180,E1 -460.713,E2 -460.713} C_VEL
LIN {X 0,Y 608.493,Z 324.088,A -85,B 0,C 180,E1 -461.186,E2 -461.186} C_VEL
LIN {X 0,Y 608.55,Z 311.285,A -85,B 0,C 180,E1 -461.554,E2 -461.554} C_VEL
LIN {X 0,Y 608.443,Z 299.532,A -85,B 0,C 180,E1 -461.788,E2 -461.788} C_VEL
LIN {X 0,Y 608.431,Z 289.437,A -85,B 0,C 180,E1 -464.379,E2 -464.379} C_VEL
LIN {X 0,Y 608.447,Z 278.846,A -85,B 0,C 180,E1 -467.13,E2 -467.13} C_VEL
LIN {X 0,Y 608.458,Z 269.579,A -85,B 0,C 180,E1 -469.57,E2 -469.57} C_VEL
LIN {X 0,Y 608.462,Z 258.726,A -85,B 0,C 180,E1 -472.476,E2 -472.476} C_VEL
LIN {X 0,Y 608.445,Z 249.72,A -85,B 0,C 180,E1 -474.935,E2 -474.935} C_VEL
LIN {X 0,Y 608.507,Z 240.453,A -85,B 0,C 180,E1 -477.515,E2 -477.515} C_VEL
LIN {X 0,Y 608.478,Z 231.837,A -85,B 0,C 180,E1 -479.972,E2 -479.972} C_VEL
LIN {X 0,Y 608.471,Z 223.114,A -85,B 0,C 180,E1 -482.523,E2 -482.523} C_VEL
LIN {X 0,Y 608.555,Z 213.975,A -85,B 0,C 180,E1 -485.27,E2 -485.27} C_VEL
LIN {X 0,Y 608.48,Z 212.693,A -85,B 0,C 180,E1 -485.681,E2 -485.681} C_VEL
LIN {X 0,Y 608.466,Z 212.696,A -85,B 0,C 180,E1 -488.239,E2 -488.239} C_VEL
LIN {X 0,Y 608.466,Z 212.696,A -85,B 0,C 180,E1 -491.342,E2 -491.342} C_VEL
LIN {X 0,Y 608.463,Z 212.694,A -85,B 0,C 180,E1 -493.869,E2 -493.869} C_VEL
LIN {X 0,Y 608.48,Z 212.694,A -85,B 0,C 180,E1 -496.689,E2 -496.689} C_VEL
LIN {X 0,Y 608.453,Z 212.698,A -85,B 0,C 180,E1 -499.696,E2 -499.696} C_VEL
LIN {X 0,Y 608.471,Z 212.693,A -85,B 0,C 180,E1 -502.253,E2 -502.253} C_VEL
LIN {X 0,Y 608.454,Z 212.697,A -85,B 0,C 180,E1 -505.093,E2 -505.093} C_VEL
LIN {X 0,Y 608.459,Z 212.696,A -85,B 0,C 180,E1 -507.904,E2 -507.904} C_VEL
LIN {X 0,Y 608.479,Z 212.694,A -85,B 0,C 180,E1 -510.22,E2 -510.22} C_VEL
LIN {X 0,Y 608.453,Z 212.698,A -85,B 0,C 180,E1 -513.225,E2 -513.225} C_VEL
LIN {X 0,Y 608.471,Z 212.693,A -85,B 0,C 180,E1 -515.847,E2 -515.847} C_VEL
LIN {X 0,Y 608.47,Z 212.695,A -85,B 0,C 180,E1 -518.308,E2 -518.308} C_VEL
LIN {X 0,Y 608.472,Z 212.693,A -85,B 0,C 180,E1 -521.282,E2 -521.282} C_VEL
LIN {X 0,Y 608.457,Z 212.696,A -85,B 0,C 180,E1 -523.905,E2 -523.905} C_VEL
LIN {X 0,Y 608.47,Z 212.695,A -85,B 0,C 180,E1 -526.643,E2 -526.643} C_VEL
LIN {X 0,Y 608.454,Z 212.695,A -85,B 0,C 180,E1 -529.349,E2 -529.349} C_VEL
LIN {X 0,Y 608.481,Z 212.694,A -85,B 0,C 180,E1 -532.032,E2 -532.032} C_VEL
LIN {X 0,Y 608.474,Z 212.693,A -85,B 0,C 180,E1 -534.697,E2 -534.697} C_VEL
LIN {X 0,Y 608.475,Z 212.694,A -85,B 0,C 180,E1 -537.351,E2 -537.351} C_VEL
LIN {X 0,Y 608.469,Z 212.694,A -85,B 0,C 180,E1 -539.999,E2 -539.999} C_VEL
LIN {X 0,Y 608.478,Z 212.693,A -85,B 0,C 180,E1 -542.647,E2 -542.647} C_VEL
LIN {X 0,Y 608.46,Z 212.696,A -85,B 0,C 180,E1 -545.301,E2 -545.301} C_VEL
LIN {X 0,Y 608.479,Z 212.692,A -85,B 0,C 180,E1 -547.966,E2 -547.966} C_VEL
LIN {X 0,Y 608.454,Z 212.695,A -85,B 0,C 180,E1 -549.466,E2 -549.466} C_VEL
LIN {X 0,Y 607.779,Z 212.782,A -85,B 0,C 180,E1 -550.02,E2 -550.02} C_VEL
LIN {X 0,Y 604.909,Z 213.138,A -85,B 0,C 180,E1 -550.917,E2 -550.917} C_VEL
LIN {X 0,Y 602.487,Z 213.483,A -85,B 0,C 180,E1 -551.638,E2 -551.638} C_VEL
LIN {X 0,Y 601.444,Z 213.927,A -85,B 0,C 180,E1 -552.193,E2 -552.193} C_VEL
LIN {X 0,Y 601.358,Z 214.14,A -85,B 0,C 180,E1 -552.38,E2 -552.38} C_VEL
LIN {X 0,Y 601.366,Z 217.223,A -85,B 0,C 180,E1 -554.897,E2 -554.897} C_VEL
LIN {X 0,Y 601.384,Z 220.529,A -85,B 0,C 180,E1 -557.687,E2 -557.687} C_VEL
LIN {X 0,Y 601.34,Z 223.859,A -85,B 0,C 180,E1 -560.524,E2 -560.524} C_VEL
LIN {X 0,Y 601.307,Z 227.618,A -85,B 0,C 180,E1 -563.413,E2 -563.413} C_VEL
LIN {X 0,Y 601.299,Z 230.845,A -85,B 0,C 180,E1 -565.846,E2 -565.846} C_VEL
LIN {X 0,Y 601.276,Z 234.609,A -85,B 0,C 180,E1 -568.633,E2 -568.633} C_VEL
LIN {X 0,Y 601.285,Z 237.781,A -85,B 0,C 180,E1 -570.948,E2 -570.948} C_VEL
LIN {X 0,Y 601.305,Z 241.905,A -85,B 0,C 180,E1 -573.919,E2 -573.919} C_VEL
LIN {X 0,Y 601.304,Z 243.677,A -85,B 0,C 180,E1 -575.183,E2 -575.183} C_VEL
LIN {X 0,Y 601.606,Z 248.836,A -85,B 0,C 180,E1 -575.299,E2 -575.299} C_VEL
LIN {X 0,Y 601.573,Z 261.748,A -85,B 0,C 180,E1 -575.651,E2 -575.651} C_VEL
LIN {X 0,Y 601.516,Z 273.62,A -85,B 0,C 180,E1 -576.106,E2 -576.106} C_VEL
LIN {X 0,Y 601.456,Z 285.085,A -85,B 0,C 180,E1 -576.681,E2 -576.681} C_VEL
LIN {X 0,Y 601.445,Z 296.497,A -85,B 0,C 180,E1 -577.416,E2 -577.416} C_VEL
LIN {X 0,Y 601.417,Z 307.068,A -85,B 0,C 180,E1 -578.266,E2 -578.266} C_VEL
LIN {X 0,Y 601.424,Z 315.728,A -85,B 0,C 180,E1 -579.123,E2 -579.123} C_VEL
LIN {X 0,Y 601.375,Z 324.036,A -85,B 0,C 180,E1 -580.138,E2 -580.138} C_VEL
LIN {X 0,Y 601.361,Z 331.218,A -85,B 0,C 180,E1 -581.232,E2 -581.232} C_VEL
LIN {X 0,Y 601.371,Z 336.13,A -85,B 0,C 180,E1 -582.176,E2 -582.176} C_VEL
LIN {X 0,Y 601.337,Z 340.021,A -85,B 0,C 180,E1 -583.118,E2 -583.118} C_VEL
LIN {X 0,Y 601.352,Z 342.991,A -85,B 0,C 180,E1 -584.055,E2 -584.055} C_VEL
LIN {X 0,Y 601.335,Z 345.147,A -85,B 0,C 180,E1 -585.003,E2 -585.003} C_VEL
LIN {X 0,Y 601.318,Z 345.909,A -85,B 0,C 180,E1 -585.473,E2 -585.473} C_VEL
LIN {X 0,Y 601.333,Z 346.825,A -85,B 0,C 180,E1 -586.434,E2 -586.434} C_VEL
LIN {X 0,Y 601.337,Z 346.92,A -85,B 0,C 180,E1 -587.415,E2 -587.415} C_VEL
LIN {X 0,Y 601.322,Z 346.148,A -85,B 0,C 180,E1 -588.415,E2 -588.415} C_VEL
LIN {X 0,Y 601.314,Z 344.442,A -85,B 0,C 180,E1 -589.435,E2 -589.435} C_VEL
LIN {X 0,Y 601.325,Z 341.705,A -85,B 0,C 180,E1 -590.475,E2 -590.475} C_VEL
LIN {X 0,Y 601.327,Z 337.792,A -85,B 0,C 180,E1 -591.539,E2 -591.539} C_VEL
LIN {X 0,Y 601.363,Z 332.524,A -85,B 0,C 180,E1 -592.624,E2 -592.624} C_VEL
LIN {X 0,Y 601.373,Z 325.587,A -85,B 0,C 180,E1 -593.74,E2 -593.74} C_VEL
LIN {X 0,Y 601.393,Z 317.504,A -85,B 0,C 180,E1 -594.765,E2 -594.765} C_VEL
LIN {X 0,Y 601.448,Z 308.623,A -85,B 0,C 180,E1 -595.681,E2 -595.681} C_VEL
LIN {X 0,Y 601.489,Z 298.994,A -85,B 0,C 180,E1 -596.49,E2 -596.49} C_VEL
LIN {X 0,Y 601.478,Z 287.362,A -85,B 0,C 180,E1 -597.273,E2 -597.273} C_VEL
LIN {X 0,Y 601.518,Z 275.795,A -85,B 0,C 180,E1 -597.886,E2 -597.886} C_VEL
LIN {X 0,Y 601.544,Z 264.15,A -85,B 0,C 180,E1 -598.36,E2 -598.36} C_VEL
LIN {X 0,Y 601.606,Z 250.795,A -85,B 0,C 180,E1 -598.746,E2 -598.746} C_VEL
LIN {X 0,Y 601.323,Z 243.688,A -85,B 0,C 180,E1 -598.899,E2 -598.899} C_VEL
LIN {X 0,Y 601.324,Z 240.236,A -85,B 0,C 180,E1 -601.368,E2 -601.368} C_VEL
LIN {X 0,Y 601.325,Z 236.399,A -85,B 0,C 180,E1 -604.146,E2 -604.146} C_VEL
LIN {X 0,Y 601.331,Z 233.073,A -85,B 0,C 180,E1 -606.587,E2 -606.587} C_VEL
LIN {X 0,Y 601.342,Z 229.202,A -85,B 0,C 180,E1 -609.476,E2 -609.476} C_VEL
LIN {X 0,Y 601.31,Z 225.484,A -85,B 0,C 180,E1 -612.309,E2 -612.309} C_VEL
LIN {X 0,Y 601.307,Z 222.88,A -85,B 0,C 180,E1 -614.406,E2 -614.406} C_VEL
LIN {X 0,Y 601.313,Z 220.341,A -85,B 0,C 180,E1 -616.482,E2 -616.482} C_VEL
LIN {X 0,Y 601.387,Z 217.045,A -85,B 0,C 180,E1 -619.224,E2 -619.224} C_VEL
LIN {X 0,Y 601.382,Z 213.749,A -85,B 0,C 180,E1 -621.939,E2 -621.939} C_VEL
LIN {X 0,Y 601.397,Z 213.573,A -85,B 0,C 180,E1 -623.963,E2 -623.963} C_VEL
LIN {X 0,Y 601.419,Z 213.571,A -85,B 0,C 180,E1 -626.651,E2 -626.651} C_VEL
LIN {X 0,Y 601.453,Z 213.569,A -85,B 0,C 180,E1 -629.331,E2 -629.331} C_VEL
LIN {X 0,Y 601.425,Z 213.572,A -85,B 0,C 180,E1 -632.009,E2 -632.009} C_VEL
LIN {X 0,Y 601.423,Z 213.57,A -85,B 0,C 180,E1 -634.692,E2 -634.692} C_VEL
LIN {X 0,Y 601.443,Z 213.568,A -85,B 0,C 180,E1 -637.385,E2 -637.385} C_VEL
LIN {X 0,Y 601.425,Z 213.573,A -85,B 0,C 180,E1 -640.095,E2 -640.095} C_VEL
LIN {X 0,Y 601.42,Z 213.572,A -85,B 0,C 180,E1 -642.828,E2 -642.828} C_VEL
LIN {X 0,Y 601.407,Z 213.572,A -85,B 0,C 180,E1 -645.592,E2 -645.592} C_VEL
LIN {X 0,Y 601.413,Z 213.574,A -85,B 0,C 180,E1 -648.392,E2 -648.392} C_VEL
LIN {X 0,Y 601.4,Z 213.574,A -85,B 0,C 180,E1 -651.24,E2 -651.24} C_VEL
LIN {X 0,Y 601.412,Z 213.574,A -85,B 0,C 180,E1 -653.411,E2 -653.411} C_VEL
LIN {X 0,Y 601.404,Z 213.573,A -85,B 0,C 180,E1 -656.364,E2 -656.364} C_VEL
LIN {X 0,Y 601.438,Z 213.568,A -85,B 0,C 180,E1 -658.793,E2 -658.793} C_VEL
LIN {X 0,Y 601.41,Z 213.574,A -85,B 0,C 180,E1 -661.727,E2 -661.727} C_VEL
LIN {X 0,Y 601.423,Z 213.573,A -85,B 0,C 180,E1 -664.119,E2 -664.119} C_VEL
LIN {X 0,Y 601.392,Z 213.576,A -85,B 0,C 180,E1 -666.584,E2 -666.584} C_VEL
LIN {X 0,Y 601.426,Z 213.57,A -85,B 0,C 180,E1 -669.126,E2 -669.126} C_VEL
LIN {X 0,Y 601.416,Z 213.571,A -85,B 0,C 180,E1 -671.766,E2 -671.766} C_VEL
LIN {X 0,Y 601.414,Z 213.573,A -85,B 0,C 180,E1 -674.537,E2 -674.537} C_VEL
LIN {X 0,Y 601.405,Z 213.574,A -85,B 0,C 180,E1 -677.331,E2 -677.331} C_VEL
LIN {X 0,Y 601.411,Z 213.572,A -85,B 0,C 180,E1 -680.007,E2 -680.007} C_VEL
LIN {X 0,Y 601.431,Z 213.569,A -85,B 0,C 180,E1 -682.619,E2 -682.619} C_VEL
LIN {X 0,Y 601.404,Z 213.573,A -85,B 0,C 180,E1 -685.069,E2 -685.069} C_VEL
LIN {X 0,Y 601.421,Z 213.571,A -85,B 0,C 180,E1 -687.486,E2 -687.486} C_VEL
LIN {X 0,Y 601.445,Z 213.568,A -85,B 0,C 180,E1 -689.849,E2 -689.849} C_VEL
LIN {X 0,Y 601.412,Z 213.575,A -85,B 0,C 180,E1 -692.638,E2 -692.638} C_VEL
LIN {X 0,Y 601.402,Z 213.575,A -85,B 0,C 180,E1 -695.123,E2 -695.123} C_VEL
LIN {X 0,Y 601.412,Z 213.575,A -85,B 0,C 180,E1 -697.396,E2 -697.396} C_VEL
LIN {X 0,Y 601.402,Z 213.573,A -85,B 0,C 180,E1 -700.192,E2 -700.192} C_VEL
LIN {X 0,Y 601.43,Z 213.57,A -85,B 0,C 180,E1 -703.016,E2 -703.016} C_VEL
LIN {X 0,Y 601.419,Z 213.572,A -85,B 0,C 180,E1 -705.91,E2 -705.91} C_VEL
LIN {X 0,Y 601.412,Z 213.572,A -85,B 0,C 180,E1 -708.543,E2 -708.543} C_VEL
LIN {X 0,Y 601.41,Z 213.572,A -85,B 0,C 180,E1 -711.263,E2 -711.263} C_VEL
LIN {X 0,Y 601.42,Z 213.573,A -85,B 0,C 180,E1 -713.964,E2 -713.964} C_VEL
LIN {X 0,Y 601.425,Z 213.571,A -85,B 0,C 180,E1 -716.652,E2 -716.652} C_VEL
LIN {X 0,Y 601.454,Z 213.566,A -85,B 0,C 180,E1 -719.332,E2 -719.332} C_VEL
LIN {X 0,Y 601.421,Z 213.571,A -85,B 0,C 180,E1 -722.01,E2 -722.01} C_VEL
LIN {X 0,Y 601.421,Z 213.573,A -85,B 0,C 180,E1 -724.693,E2 -724.693} C_VEL
LIN {X 0,Y 601.445,Z 213.569,A -85,B 0,C 180,E1 -727.386,E2 -727.386} C_VEL
LIN {X 0,Y 601.424,Z 213.57,A -85,B 0,C 180,E1 -730.096,E2 -730.096} C_VEL
LIN {X 0,Y 601.414,Z 213.572,A -85,B 0,C 180,E1 -732.829,E2 -732.829} C_VEL
LIN {X 0,Y 601.412,Z 213.574,A -85,B 0,C 180,E1 -735.592,E2 -735.592} C_VEL
LIN {X 0,Y 601.403,Z 213.574,A -85,B 0,C 180,E1 -737.689,E2 -737.689} C_VEL
LIN {X 0,Y 601.431,Z 213.57,A -85,B 0,C 180,E1 -740.523,E2 -740.523} C_VEL
LIN {X 0,Y 601.423,Z 213.57,A -85,B 0,C 180,E1 -743.411,E2 -743.411} C_VEL
LIN {X 0,Y 601.402,Z 213.575,A -85,B 0,C 180,E1 -746.365,E2 -746.365} C_VEL
LIN {X 0,Y 601.441,Z 213.57,A -85,B 0,C 180,E1 -748.789,E2 -748.789} C_VEL
LIN {X 0,Y 601.403,Z 213.573,A -85,B 0,C 180,E1 -751.728,E2 -751.728} C_VEL
LIN {X 0,Y 601.424,Z 213.57,A -85,B 0,C 180,E1 -754.119,E2 -754.119} C_VEL
LIN {X 0,Y 601.405,Z 213.573,A -85,B 0,C 180,E1 -756.584,E2 -756.584} C_VEL
LIN {X 0,Y 601.417,Z 213.572,A -85,B 0,C 180,E1 -759.127,E2 -759.127} C_VEL
LIN {X 0,Y 601.421,Z 213.574,A -85,B 0,C 180,E1 -761.766,E2 -761.766} C_VEL
LIN {X 0,Y 601.431,Z 213.569,A -85,B 0,C 180,E1 -764.535,E2 -764.535} C_VEL
LIN {X 0,Y 601.418,Z 213.572,A -85,B 0,C 180,E1 -767.409,E2 -767.409} C_VEL
LIN {X 0,Y 601.445,Z 213.568,A -85,B 0,C 180,E1 -770.464,E2 -770.464} C_VEL
LIN {X 0,Y 601.399,Z 213.575,A -85,B 0,C 180,E1 -773.417,E2 -773.417} C_VEL
LIN {X 0,Y 601.431,Z 213.685,A -85,B 0,C 180,E1 -774.158,E2 -774.158} C_VEL
LIN {X 0,Y 601.579,Z 220.851,A -85,B 0,C 180,E1 -776.373,E2 -776.373} C_VEL
LIN {X 0,Y 601.498,Z 229.859,A -85,B 0,C 180,E1 -779.062,E2 -779.062} C_VEL
LIN {X 0,Y 601.462,Z 237.802,A -85,B 0,C 180,E1 -781.374,E2 -781.374} C_VEL
LIN {X 0,Y 601.482,Z 247.451,A -85,B 0,C 180,E1 -784.12,E2 -784.12} C_VEL
LIN {X 0,Y 601.46,Z 256.337,A -85,B 0,C 180,E1 -786.591,E2 -786.591} C_VEL
LIN {X 0,Y 601.432,Z 266.928,A -85,B 0,C 180,E1 -789.478,E2 -789.478} C_VEL
LIN {X 0,Y 601.405,Z 277.519,A -85,B 0,C 180,E1 -792.312,E2 -792.312} C_VEL
LIN {X 0,Y 601.368,Z 288.11,A -85,B 0,C 180,E1 -795.101,E2 -795.101} C_VEL
LIN {X 0,Y 601.351,Z 298.702,A -85,B 0,C 180,E1 -797.856,E2 -797.856} C_VEL
LIN {X 0,Y 601.38,Z 299.529,A -85,B 0,C 180,E1 -798.07,E2 -798.07} C_VEL
LIN {X 0,Y 601.602,Z 312.168,A -85,B 0,C 180,E1 -798.331,E2 -798.331} C_VEL
LIN {X 0,Y 601.535,Z 324.333,A -85,B 0,C 180,E1 -798.691,E2 -798.691} C_VEL
LIN {X 0,Y 601.484,Z 335.223,A -85,B 0,C 180,E1 -799.131,E2 -799.131} C_VEL
LIN {X 0,Y 601.483,Z 346.75,A -85,B 0,C 180,E1 -799.735,E2 -799.735} C_VEL
LIN {X 0,Y 601.462,Z 358.248,A -85,B 0,C 180,E1 -800.5,E2 -800.5} C_VEL
LIN {X 0,Y 601.436,Z 367.533,A -85,B 0,C 180,E1 -801.262,E2 -801.262} C_VEL
LIN {X 0,Y 601.401,Z 375.986,A -85,B 0,C 180,E1 -802.107,E2 -802.107} C_VEL
LIN {X 0,Y 601.382,Z 384.233,A -85,B 0,C 180,E1 -803.12,E2 -803.12} C_VEL
LIN {X 0,Y 601.373,Z 390.875,A -85,B 0,C 180,E1 -804.13,E2 -804.13} C_VEL
LIN {X 0,Y 601.336,Z 396.949,A -85,B 0,C 180,E1 -805.307,E2 -805.307} C_VEL
LIN {X 0,Y 601.368,Z 400.895,A -85,B 0,C 180,E1 -806.314,E2 -806.314} C_VEL
LIN {X 0,Y 601.325,Z 403.808,A -85,B 0,C 180,E1 -807.32,E2 -807.32} C_VEL
LIN {X 0,Y 601.343,Z 405.201,A -85,B 0,C 180,E1 -807.99,E2 -807.99} C_VEL
LIN {X 0,Y 601.339,Z 406.783,A -85,B 0,C 180,E1 -809.33,E2 -809.33} C_VEL
LIN {X 0,Y 601.335,Z 407,A -85,B 0,C 180,E1 -810,E2 -810} C_VEL
LIN {X 0,Y 601.347,Z 406.184,A -85,B 0,C 180,E1 -811.339,E2 -811.339} C_VEL
LIN {X 0,Y 601.343,Z 405.202,A -85,B 0,C 180,E1 -812.009,E2 -812.009} C_VEL
LIN {X 0,Y 601.325,Z 403.81,A -85,B 0,C 180,E1 -812.679,E2 -812.679} C_VEL
LIN {X 0,Y 601.368,Z 400.897,A -85,B 0,C 180,E1 -813.685,E2 -813.685} C_VEL
LIN {X 0,Y 601.336,Z 396.952,A -85,B 0,C 180,E1 -814.692,E2 -814.692} C_VEL
LIN {X 0,Y 601.373,Z 390.879,A -85,B 0,C 180,E1 -815.869,E2 -815.869} C_VEL
LIN {X 0,Y 601.382,Z 384.238,A -85,B 0,C 180,E1 -816.879,E2 -816.879} C_VEL
LIN {X 0,Y 601.4,Z 375.993,A -85,B 0,C 180,E1 -817.892,E2 -817.892} C_VEL
LIN {X 0,Y 601.436,Z 367.541,A -85,B 0,C 180,E1 -818.737,E2 -818.737} C_VEL
LIN {X 0,Y 601.451,Z 357.097,A -85,B 0,C 180,E1 -819.585,E2 -819.585} C_VEL
LIN {X 0,Y 601.483,Z 346.763,A -85,B 0,C 180,E1 -820.264,E2 -820.264} C_VEL
LIN {X 0,Y 601.484,Z 335.224,A -85,B 0,C 180,E1 -820.869,E2 -820.869} C_VEL
LIN {X 0,Y 601.527,Z 322.345,A -85,B 0,C 180,E1 -821.375,E2 -821.375} C_VEL
LIN {X 0,Y 601.617,Z 309.457,A -85,B 0,C 180,E1 -821.732,E2 -821.732} C_VEL
LIN {X 0,Y 601.38,Z 299.532,A -85,B 0,C 180,E1 -821.929,E2 -821.929} C_VEL
LIN {X 0,Y 601.381,Z 289.437,A -85,B 0,C 180,E1 -824.552,E2 -824.552} C_VEL
LIN {X 0,Y 601.393,Z 278.846,A -85,B 0,C 180,E1 -827.337,E2 -827.337} C_VEL
LIN {X 0,Y 601.426,Z 268.255,A -85,B 0,C 180,E1 -830.164,E2 -830.164} C_VEL
LIN {X 0,Y 601.43,Z 258.988,A -85,B 0,C 180,E1 -832.682,E2 -832.682} C_VEL
LIN {X 0,Y 601.446,Z 249.72,A -85,B 0,C 180,E1 -835.246,E2 -835.246} C_VEL
LIN {X 0,Y 601.502,Z 240.453,A -85,B 0,C 180,E1 -837.863,E2 -837.863} C_VEL
LIN {X 0,Y 601.471,Z 231.186,A -85,B 0,C 180,E1 -840.549,E2 -840.549} C_VEL
LIN {X 0,Y 601.508,Z 223.844,A -85,B 0,C 180,E1 -842.727,E2 -842.727} C_VEL
LIN {X 0,Y 601.585,Z 215.921,A -85,B 0,C 180,E1 -845.137,E2 -845.137} C_VEL
LIN {X 0,Y 601.426,Z 213.573,A -85,B 0,C 180,E1 -845.931,E2 -845.931} C_VEL
LIN {X 0,Y 601.416,Z 213.573,A -85,B 0,C 180,E1 -848.468,E2 -848.468} C_VEL
LIN {X 0,Y 601.415,Z 213.572,A -85,B 0,C 180,E1 -850.874,E2 -850.874} C_VEL
LIN {X 0,Y 601.43,Z 213.572,A -85,B 0,C 180,E1 -853.585,E2 -853.585} C_VEL
LIN {X 0,Y 601.43,Z 213.571,A -85,B 0,C 180,E1 -856.426,E2 -856.426} C_VEL
LIN {X 0,Y 601.419,Z 213.572,A -85,B 0,C 180,E1 -859.425,E2 -859.425} C_VEL
LIN {X 0,Y 601.426,Z 213.573,A -85,B 0,C 180,E1 -861.732,E2 -861.732} C_VEL
LIN {X 0,Y 601.387,Z 213.576,A -85,B 0,C 180,E1 -864.245,E2 -864.245} C_VEL
LIN {X 0,Y 601.414,Z 213.573,A -85,B 0,C 180,E1 -866.685,E2 -866.685} C_VEL
LIN {X 0,Y 601.422,Z 213.574,A -85,B 0,C 180,E1 -869.057,E2 -869.057} C_VEL
LIN {X 0,Y 601.429,Z 213.571,A -85,B 0,C 180,E1 -871.372,E2 -871.372} C_VEL
LIN {X 0,Y 601.406,Z 213.573,A -85,B 0,C 180,E1 -873.636,E2 -873.636} C_VEL
LIN {X 0,Y 601.421,Z 213.572,A -85,B 0,C 180,E1 -876.589,E2 -876.589} C_VEL
LIN {X 0,Y 601.433,Z 213.572,A -85,B 0,C 180,E1 -879.477,E2 -879.477} C_VEL
LIN {X 0,Y 601.398,Z 213.574,A -85,B 0,C 180,E1 -882.311,E2 -882.311} C_VEL
LIN {X 0,Y 601.413,Z 213.573,A -85,B 0,C 180,E1 -884.408,E2 -884.408} C_VEL
LIN {X 0,Y 601.419,Z 213.572,A -85,B 0,C 180,E1 -887.171,E2 -887.171} C_VEL
LIN {X 0,Y 601.429,Z 213.573,A -85,B 0,C 180,E1 -889.904,E2 -889.904} C_VEL
LIN {X 0,Y 601.456,Z 213.567,A -85,B 0,C 180,E1 -892.614,E2 -892.614} C_VEL
LIN {X 0,Y 601.418,Z 213.573,A -85,B 0,C 180,E1 -895.307,E2 -895.307} C_VEL
LIN {X 0,Y 601.424,Z 213.572,A -85,B 0,C 180,E1 -897.99,E2 -897.99} C_VEL
LIN {X 0,Y 601.451,Z 213.568,A -85,B 0,C 180,E1 -900.668,E2 -900.668} C_VEL
LIN {X 0,Y 601.427,Z 213.573,A -85,B 0,C 180,E1 -903.348,E2 -903.348} C_VEL
LIN {X 0,Y 601.41,Z 213.573,A -85,B 0,C 180,E1 -906.036,E2 -906.036} C_VEL
LIN {X 0,Y 601.439,Z 213.571,A -85,B 0,C 180,E1 -908.736,E2 -908.736} C_VEL
LIN {X 0,Y 601.409,Z 213.573,A -85,B 0,C 180,E1 -911.457,E2 -911.457} C_VEL
LIN {X 0,Y 601.358,Z 214.14,A -85,B 0,C 180,E1 -912.38,E2 -912.38} C_VEL
LIN {X 0,Y 600.685,Z 214.89,A -85,B 0,C 180,E1 -912.935,E2 -912.935} C_VEL
LIN {X 0,Y 597.822,Z 216.254,A -85,B 0,C 180,E1 -913.834,E2 -913.834} C_VEL
LIN {X 0,Y 595.403,Z 217.351,A -85,B 0,C 180,E1 -914.557,E2 -914.557} C_VEL
LIN {X 0,Y 594.362,Z 218.108,A -85,B 0,C 180,E1 -915.115,E2 -915.115} C_VEL
LIN {X 0,Y 594.276,Z 218.341,A -85,B 0,C 180,E1 -915.305,E2 -915.305} C_VEL
LIN {X 0,Y 594.301,Z 221.424,A -85,B 0,C 180,E1 -917.905,E2 -917.905} C_VEL
LIN {X 0,Y 594.283,Z 224.741,A -85,B 0,C 180,E1 -920.778,E2 -920.778} C_VEL
LIN {X 0,Y 594.222,Z 228.391,A -85,B 0,C 180,E1 -923.71,E2 -923.71} C_VEL
LIN {X 0,Y 594.206,Z 231.384,A -85,B 0,C 180,E1 -925.988,E2 -925.988} C_VEL
LIN {X 0,Y 594.182,Z 234.381,A -85,B 0,C 180,E1 -928.235,E2 -928.235} C_VEL
LIN {X 0,Y 594.207,Z 237.532,A -85,B 0,C 180,E1 -930.568,E2 -930.568} C_VEL
LIN {X 0,Y 594.222,Z 241.919,A -85,B 0,C 180,E1 -933.769,E2 -933.769} C_VEL
LIN {X 0,Y 594.232,Z 243.679,A -85,B 0,C 180,E1 -935.041,E2 -935.041} C_VEL
LIN {X 0,Y 594.665,Z 250.094,A -85,B 0,C 180,E1 -935.189,E2 -935.189} C_VEL
LIN {X 0,Y 594.606,Z 262.634,A -85,B 0,C 180,E1 -935.545,E2 -935.545} C_VEL
LIN {X 0,Y 594.519,Z 274.65,A -85,B 0,C 180,E1 -936.021,E2 -936.021} C_VEL
LIN {X 0,Y 594.449,Z 285.421,A -85,B 0,C 180,E1 -936.577,E2 -936.577} C_VEL
LIN {X 0,Y 594.438,Z 296.09,A -85,B 0,C 180,E1 -937.272,E2 -937.272} C_VEL
LIN {X 0,Y 594.379,Z 306.989,A -85,B 0,C 180,E1 -938.154,E2 -938.154} C_VEL
LIN {X 0,Y 594.347,Z 315.684,A -85,B 0,C 180,E1 -939.023,E2 -939.023} C_VEL
LIN {X 0,Y 594.312,Z 323.142,A -85,B 0,C 180,E1 -939.932,E2 -939.932} C_VEL
LIN {X 0,Y 594.271,Z 329.131,A -85,B 0,C 180,E1 -940.811,E2 -940.811} C_VEL
LIN {X 0,Y 594.296,Z 334.811,A -85,B 0,C 180,E1 -941.84,E2 -941.84} C_VEL
LIN {X 0,Y 594.281,Z 339.196,A -85,B 0,C 180,E1 -942.844,E2 -942.844} C_VEL
LIN {X 0,Y 594.244,Z 342.486,A -85,B 0,C 180,E1 -943.828,E2 -943.828} C_VEL
LIN {X 0,Y 594.251,Z 345.508,A -85,B 0,C 180,E1 -945.2,E2 -945.2} C_VEL
LIN {X 0,Y 594.224,Z 346.65,A -85,B 0,C 180,E1 -946.173,E2 -946.173} C_VEL
LIN {X 0,Y 594.24,Z 346.98,A -85,B 0,C 180,E1 -947.158,E2 -947.158} C_VEL
LIN {X 0,Y 594.217,Z 346.044,A -85,B 0,C 180,E1 -948.523,E2 -948.523} C_VEL
LIN {X 0,Y 594.235,Z 344.529,A -85,B 0,C 180,E1 -949.423,E2 -949.423} C_VEL
LIN {X 0,Y 594.231,Z 342.35,A -85,B 0,C 180,E1 -950.309,E2 -950.309} C_VEL
LIN {X 0,Y 594.253,Z 338.965,A -85,B 0,C 180,E1 -951.309,E2 -951.309} C_VEL
LIN {X 0,Y 594.261,Z 334.048,A -85,B 0,C 180,E1 -952.405,E2 -952.405} C_VEL
LIN {X 0,Y 594.307,Z 327.552,A -85,B 0,C 180,E1 -953.524,E2 -953.524} C_VEL
LIN {X 0,Y 594.309,Z 319.779,A -85,B 0,C 180,E1 -954.589,E2 -954.589} C_VEL
LIN {X 0,Y 594.388,Z 311.099,A -85,B 0,C 180,E1 -955.546,E2 -955.546} C_VEL
LIN {X 0,Y 594.438,Z 300.97,A -85,B 0,C 180,E1 -956.447,E2 -956.447} C_VEL
LIN {X 0,Y 594.46,Z 291.463,A -85,B 0,C 180,E1 -957.137,E2 -957.137} C_VEL
LIN {X 0,Y 594.515,Z 280.87,A -85,B 0,C 180,E1 -957.762,E2 -957.762} C_VEL
LIN {X 0,Y 594.59,Z 268.724,A -85,B 0,C 180,E1 -958.321,E2 -958.321} C_VEL
LIN {X 0,Y 594.639,Z 255.469,A -85,B 0,C 180,E1 -958.765,E2 -958.765} C_VEL
LIN {X 0,Y 594.477,Z 245.421,A -85,B 0,C 180,E1 -959.003,E2 -959.003} C_VEL
LIN {X 0,Y 594.226,Z 243.66,A -85,B 0,C 180,E1 -959.063,E2 -959.063} C_VEL
LIN {X 0,Y 594.216,Z 239.931,A -85,B 0,C 180,E1 -961.765,E2 -961.765} C_VEL
LIN {X 0,Y 594.229,Z 236.815,A -85,B 0,C 180,E1 -964.05,E2 -964.05} C_VEL
LIN {X 0,Y 594.234,Z 233.795,A -85,B 0,C 180,E1 -966.29,E2 -966.29} C_VEL
LIN {X 0,Y 594.287,Z 229.905,A -85,B 0,C 180,E1 -969.221,E2 -969.221} C_VEL
LIN {X 0,Y 594.217,Z 226.178,A -85,B 0,C 180,E1 -972.091,E2 -972.091} C_VEL
LIN {X 0,Y 594.239,Z 223.719,A -85,B 0,C 180,E1 -974.216,E2 -974.216} C_VEL
LIN {X 0,Y 594.244,Z 221.125,A -85,B 0,C 180,E1 -976.318,E2 -976.318} C_VEL
LIN {X 0,Y 594.315,Z 217.78,A -85,B 0,C 180,E1 -979.094,E2 -979.094} C_VEL
LIN {X 0,Y 594.302,Z 214.477,A -85,B 0,C 180,E1 -981.842,E2 -981.842} C_VEL
LIN {X 0,Y 594.353,Z 214.451,A -85,B 0,C 180,E1 -983.891,E2 -983.891} C_VEL
LIN {X 0,Y 594.371,Z 214.448,A -85,B 0,C 180,E1 -986.611,E2 -986.611} C_VEL
LIN {X 0,Y 594.422,Z 214.445,A -85,B 0,C 180,E1 -989.323,E2 -989.323} C_VEL
LIN {X 0,Y 594.393,Z 214.447,A -85,B 0,C 180,E1 -992.033,E2 -992.033} C_VEL
LIN {X 0,Y 594.392,Z 214.446,A -85,B 0,C 180,E1 -994.748,E2 -994.748} C_VEL
LIN {X 0,Y 594.407,Z 214.445,A -85,B 0,C 180,E1 -997.473,E2 -997.473} C_VEL
LIN {X 0,Y 594.386,Z 214.45,A -85,B 0,C 180,E1 -1000.216,E2 -1000.216} C_VEL
LIN {X 0,Y 594.365,Z 214.45,A -85,B 0,C 180,E1 -1002.983,E2 -1002.983} C_VEL
LIN {X 0,Y 594.362,Z 214.45,A -85,B 0,C 180,E1 -1005.781,E2 -1005.781} C_VEL
LIN {X 0,Y 594.379,Z 214.45,A -85,B 0,C 180,E1 -1008.618,E2 -1008.618} C_VEL
LIN {X 0,Y 594.36,Z 214.45,A -85,B 0,C 180,E1 -1011.504,E2 -1011.504} C_VEL
LIN {X 0,Y 594.379,Z 214.447,A -85,B 0,C 180,E1 -1013.705,E2 -1013.705} C_VEL
LIN {X 0,Y 594.38,Z 214.449,A -85,B 0,C 180,E1 -1016.7,E2 -1016.7} C_VEL
LIN {X 0,Y 594.376,Z 214.449,A -85,B 0,C 180,E1 -1018.999,E2 -1018.999} C_VEL
LIN {X 0,Y 594.384,Z 214.45,A -85,B 0,C 180,E1 -1021.647,E2 -1021.647} C_VEL
LIN {X 0,Y 594.387,Z 214.446,A -85,B 0,C 180,E1 -1024.58,E2 -1024.58} C_VEL
LIN {X 0,Y 594.38,Z 214.451,A -85,B 0,C 180,E1 -1027.61,E2 -1027.61} C_VEL
LIN {X 0,Y 594.38,Z 214.447,A -85,B 0,C 180,E1 -1030.566,E2 -1030.566} C_VEL
LIN {X 0,Y 594.376,Z 214.449,A -85,B 0,C 180,E1 -1033.299,E2 -1033.299} C_VEL
LIN {X 0,Y 594.374,Z 214.45,A -85,B 0,C 180,E1 -1036.16,E2 -1036.16} C_VEL
LIN {X 0,Y 594.377,Z 214.449,A -85,B 0,C 180,E1 -1039.178,E2 -1039.178} C_VEL
LIN {X 0,Y 594.384,Z 214.449,A -85,B 0,C 180,E1 -1042.061,E2 -1042.061} C_VEL
LIN {X 0,Y 594.351,Z 214.451,A -85,B 0,C 180,E1 -1044.677,E2 -1044.677} C_VEL
LIN {X 0,Y 594.373,Z 214.448,A -85,B 0,C 180,E1 -1047.09,E2 -1047.09} C_VEL
LIN {X 0,Y 594.397,Z 214.445,A -85,B 0,C 180,E1 -1049.671,E2 -1049.671} C_VEL
LIN {X 0,Y 594.37,Z 214.452,A -85,B 0,C 180,E1 -1052.541,E2 -1052.541} C_VEL
LIN {X 0,Y 594.372,Z 214.45,A -85,B 0,C 180,E1 -1054.808,E2 -1054.808} C_VEL
LIN {X 0,Y 594.361,Z 214.452,A -85,B 0,C 180,E1 -1057.266,E2 -1057.266} C_VEL
LIN {X 0,Y 594.37,Z 214.45,A -85,B 0,C 180,E1 -1059.948,E2 -1059.948} C_VEL
LIN {X 0,Y 594.387,Z 214.446,A -85,B 0,C 180,E1 -1062.808,E2 -1062.808} C_VEL
LIN {X 0,Y 594.387,Z 214.449,A -85,B 0,C 180,E1 -1065.828,E2 -1065.828} C_VEL
LIN {X 0,Y 594.38,Z 214.448,A -85,B 0,C 180,E1 -1068.405,E2 -1068.405} C_VEL
LIN {X 0,Y 594.377,Z 214.448,A -85,B 0,C 180,E1 -1071.159,E2 -1071.159} C_VEL
LIN {X 0,Y 594.376,Z 214.45,A -85,B 0,C 180,E1 -1073.892,E2 -1073.892} C_VEL
LIN {X 0,Y 594.376,Z 214.45,A -85,B 0,C 180,E1 -1076.612,E2 -1076.612} C_VEL
LIN {X 0,Y 594.425,Z 214.442,A -85,B 0,C 180,E1 -1079.324,E2 -1079.324} C_VEL
LIN {X 0,Y 594.392,Z 214.447,A -85,B 0,C 180,E1 -1082.034,E2 -1082.034} C_VEL
LIN {X 0,Y 594.391,Z 214.449,A -85,B 0,C 180,E1 -1084.749,E2 -1084.749} C_VEL
LIN {X 0,Y 594.397,Z 214.446,A -85,B 0,C 180,E1 -1087.474,E2 -1087.474} C_VEL
LIN {X 0,Y 594.387,Z 214.447,A -85,B 0,C 180,E1 -1090.217,E2 -1090.217} C_VEL
LIN {X 0,Y 594.363,Z 214.451,A -85,B 0,C 180,E1 -1092.984,E2 -1092.984} C_VEL
LIN {X 0,Y 594.375,Z 214.448,A -85,B 0,C 180,E1 -1095.079,E2 -1095.079} C_VEL
LIN {X 0,Y 594.396,Z 214.446,A -85,B 0,C 180,E1 -1097.194,E2 -1097.194} C_VEL
LIN {X 0,Y 594.375,Z 214.45,A -85,B 0,C 180,E1 -1100.055,E2 -1100.055} C_VEL
LIN {X 0,Y 594.37,Z 214.45,A -85,B 0,C 180,E1 -1102.968,E2 -1102.968} C_VEL
LIN {X 0,Y 594.363,Z 214.452,A -85,B 0,C 180,E1 -1105.194,E2 -1105.194} C_VEL
LIN {X 0,Y 594.392,Z 214.449,A -85,B 0,C 180,E1 -1107.527,E2 -1107.527} C_VEL
LIN {X 0,Y 594.373,Z 214.448,A -85,B 0,C 180,E1 -1110.326,E2 -1110.326} C_VEL
LIN {X 0,Y 594.383,Z 214.447,A -85,B 0,C 180,E1 -1112.951,E2 -1112.951} C_VEL
LIN {X 0,Y 594.358,Z 214.451,A -85,B 0,C 180,E1 -1115.409,E2 -1115.409} C_VEL
LIN {X 0,Y 594.392,Z 214.447,A -85,B 0,C 180,E1 -1117.941,E2 -1117.941} C_VEL
LIN {X 0,Y 594.377,Z 214.449,A -85,B 0,C 180,E1 -1120.822,E2 -1120.822} C_VEL
LIN {X 0,Y 594.373,Z 214.449,A -85,B 0,C 180,E1 -1123.84,E2 -1123.84} C_VEL
LIN {X 0,Y 594.372,Z 214.45,A -85,B 0,C 180,E1 -1126.701,E2 -1126.701} C_VEL
LIN {X 0,Y 594.367,Z 214.449,A -85,B 0,C 180,E1 -1129.433,E2 -1129.433} C_VEL
LIN {X 0,Y 594.39,Z 214.449,A -85,B 0,C 180,E1 -1132.392,E2 -1132.392} C_VEL
LIN {X 0,Y 594.398,Z 214.634,A -85,B 0,C 180,E1 -1133.968,E2 -1133.968} C_VEL
LIN {X 0,Y 594.609,Z 219.268,A -85,B 0,C 180,E1 -1135.435,E2 -1135.435} C_VEL
LIN {X 0,Y 594.54,Z 225.887,A -85,B 0,C 180,E1 -1137.462,E2 -1137.462} C_VEL
LIN {X 0,Y 594.514,Z 233.194,A -85,B 0,C 180,E1 -1139.652,E2 -1139.652} C_VEL
LIN {X 0,Y 594.506,Z 243.098,A -85,B 0,C 180,E1 -1142.545,E2 -1142.545} C_VEL
LIN {X 0,Y 594.459,Z 252.365,A -85,B 0,C 180,E1 -1145.184,E2 -1145.184} C_VEL
LIN {X 0,Y 594.413,Z 262.956,A -85,B 0,C 180,E1 -1148.134,E2 -1148.134} C_VEL
LIN {X 0,Y 594.363,Z 273.747,A -85,B 0,C 180,E1 -1151.078,E2 -1151.078} C_VEL
LIN {X 0,Y 594.315,Z 284.139,A -85,B 0,C 180,E1 -1153.865,E2 -1153.865} C_VEL
LIN {X 0,Y 594.325,Z 294.73,A -85,B 0,C 180,E1 -1156.668,E2 -1156.668} C_VEL
LIN {X 0,Y 594.291,Z 299.529,A -85,B 0,C 180,E1 -1157.926,E2 -1157.926} C_VEL
LIN {X 0,Y 594.674,Z 305.213,A -85,B 0,C 180,E1 -1158.042,E2 -1158.042} C_VEL
LIN {X 0,Y 594.617,Z 318.484,A -85,B 0,C 180,E1 -1158.365,E2 -1158.365} C_VEL
LIN {X 0,Y 594.533,Z 330.626,A -85,B 0,C 180,E1 -1158.8,E2 -1158.8} C_VEL
LIN {X 0,Y 594.479,Z 342.201,A -85,B 0,C 180,E1 -1159.355,E2 -1159.355} C_VEL
LIN {X 0,Y 594.471,Z 353.471,A -85,B 0,C 180,E1 -1160.043,E2 -1160.043} C_VEL
LIN {X 0,Y 594.406,Z 363.643,A -85,B 0,C 180,E1 -1160.815,E2 -1160.815} C_VEL
LIN {X 0,Y 594.373,Z 372.784,A -85,B 0,C 180,E1 -1161.671,E2 -1161.671} C_VEL
LIN {X 0,Y 594.317,Z 381.688,A -85,B 0,C 180,E1 -1162.696,E2 -1162.696} C_VEL
LIN {X 0,Y 594.281,Z 388.172,A -85,B 0,C 180,E1 -1163.615,E2 -1163.615} C_VEL
LIN {X 0,Y 594.289,Z 393.678,A -85,B 0,C 180,E1 -1164.571,E2 -1164.571} C_VEL
LIN {X 0,Y 594.27,Z 398.37,A -85,B 0,C 180,E1 -1165.591,E2 -1165.591} C_VEL
LIN {X 0,Y 594.267,Z 401.955,A -85,B 0,C 180,E1 -1166.61,E2 -1166.61} C_VEL
LIN {X 0,Y 594.226,Z 403.808,A -85,B 0,C 180,E1 -1167.288,E2 -1167.288} C_VEL
LIN {X 0,Y 594.242,Z 405.201,A -85,B 0,C 180,E1 -1167.966,E2 -1167.966} C_VEL
LIN {X 0,Y 594.239,Z 406.783,A -85,B 0,C 180,E1 -1169.322,E2 -1169.322} C_VEL
LIN {X 0,Y 594.236,Z 407,A -85,B 0,C 180,E1 -1170,E2 -1170} C_VEL
LIN {X 0,Y 594.247,Z 406.185,A -85,B 0,C 180,E1 -1171.355,E2 -1171.355} C_VEL
LIN {X 0,Y 594.242,Z 405.202,A -85,B 0,C 180,E1 -1172.033,E2 -1172.033} C_VEL
LIN {X 0,Y 594.226,Z 403.81,A -85,B 0,C 180,E1 -1172.711,E2 -1172.711} C_VEL
LIN {X 0,Y 594.289,Z 400.897,A -85,B 0,C 180,E1 -1173.729,E2 -1173.729} C_VEL
LIN {X 0,Y 594.241,Z 396.951,A -85,B 0,C 180,E1 -1174.748,E2 -1174.748} C_VEL
LIN {X 0,Y 594.305,Z 390.879,A -85,B 0,C 180,E1 -1175.939,E2 -1175.939} C_VEL
LIN {X 0,Y 594.308,Z 384.238,A -85,B 0,C 180,E1 -1176.962,E2 -1176.962} C_VEL
LIN {X 0,Y 594.359,Z 375.993,A -85,B 0,C 180,E1 -1177.986,E2 -1177.986} C_VEL
LIN {X 0,Y 594.382,Z 367.541,A -85,B 0,C 180,E1 -1178.842,E2 -1178.842} C_VEL
LIN {X 0,Y 594.435,Z 357.098,A -85,B 0,C 180,E1 -1179.699,E2 -1179.699} C_VEL
LIN {X 0,Y 594.459,Z 346.764,A -85,B 0,C 180,E1 -1180.386,E2 -1180.386} C_VEL
LIN {X 0,Y 594.502,Z 334.777,A -85,B 0,C 180,E1 -1181.019,E2 -1181.019} C_VEL
LIN {X 0,Y 594.564,Z 322.502,A -85,B 0,C 180,E1 -1181.505,E2 -1181.505} C_VEL
LIN {X 0,Y 594.678,Z 309.457,A -85,B 0,C 180,E1 -1181.871,E2 -1181.871} C_VEL
LIN {X 0,Y 594.443,Z 300.807,A -85,B 0,C 180,E1 -1182.039,E2 -1182.039} C_VEL
LIN {X 0,Y 594.291,Z 299.532,A -85,B 0,C 180,E1 -1182.073,E2 -1182.073} C_VEL
LIN {X 0,Y 594.31,Z 289.437,A -85,B 0,C 180,E1 -1184.729,E2 -1184.729} C_VEL
LIN {X 0,Y 594.337,Z 278.846,A -85,B 0,C 180,E1 -1187.549,E2 -1187.549} C_VEL
LIN {X 0,Y 594.384,Z 268.255,A -85,B 0,C 180,E1 -1190.414,E2 -1190.414} C_VEL
LIN {X 0,Y 594.433,Z 257.664,A -85,B 0,C 180,E1 -1193.332,E2 -1193.332} C_VEL
LIN {X 0,Y 594.488,Z 248.032,A -85,B 0,C 180,E1 -1196.042,E2 -1196.042} C_VEL
LIN {X 0,Y 594.471,Z 239.151,A -85,B 0,C 180,E1 -1198.6,E2 -1198.6} C_VEL
LIN {X 0,Y 594.529,Z 231.186,A -85,B 0,C 180,E1 -1200.945,E2 -1200.945} C_VEL
LIN {X 0,Y 594.614,Z 221.919,A -85,B 0,C 180,E1 -1203.745,E2 -1203.745} C_VEL
LIN {X 0,Y 594.569,Z 215.299,A -85,B 0,C 180,E1 -1205.81,E2 -1205.81} C_VEL
LIN {X 0,Y 594.372,Z 214.452,A -85,B 0,C 180,E1 -1206.137,E2 -1206.137} C_VEL
LIN {X 0,Y 594.372,Z 214.45,A -85,B 0,C 180,E1 -1208.805,E2 -1208.805} C_VEL
LIN {X 0,Y 594.382,Z 214.449,A -85,B 0,C 180,E1 -1211.847,E2 -1211.847} C_VEL
LIN {X 0,Y 594.364,Z 214.451,A -85,B 0,C 180,E1 -1214.808,E2 -1214.808} C_VEL
LIN {X 0,Y 594.373,Z 214.452,A -85,B 0,C 180,E1 -1217.624,E2 -1217.624} C_VEL
LIN {X 0,Y 594.39,Z 214.447,A -85,B 0,C 180,E1 -1220.32,E2 -1220.32} C_VEL
LIN {X 0,Y 594.385,Z 214.45,A -85,B 0,C 180,E1 -1222.913,E2 -1222.913} C_VEL
LIN {X 0,Y 594.383,Z 214.45,A -85,B 0,C 180,E1 -1225.86,E2 -1225.86} C_VEL
LIN {X 0,Y 594.378,Z 214.448,A -85,B 0,C 180,E1 -1228.649,E2 -1228.649} C_VEL
LIN {X 0,Y 594.383,Z 214.449,A -85,B 0,C 180,E1 -1231.041,E2 -1231.041} C_VEL
LIN {X 0,Y 594.391,Z 214.447,A -85,B 0,C 180,E1 -1233.975,E2 -1233.975} C_VEL
LIN {X 0,Y 594.388,Z 214.449,A -85,B 0,C 180,E1 -1236.295,E2 -1236.295} C_VEL
LIN {X 0,Y 594.407,Z 214.445,A -85,B 0,C 180,E1 -1239.224,E2 -1239.224} C_VEL
LIN {X 0,Y 594.354,Z 214.451,A -85,B 0,C 180,E1 -1242.094,E2 -1242.094} C_VEL
LIN {X 0,Y 594.367,Z 214.45,A -85,B 0,C 180,E1 -1244.218,E2 -1244.218} C_VEL
LIN {X 0,Y 594.367,Z 214.451,A -85,B 0,C 180,E1 -1247.016,E2 -1247.016} C_VEL
LIN {X 0,Y 594.388,Z 214.449,A -85,B 0,C 180,E1 -1249.783,E2 -1249.783} C_VEL
LIN {X 0,Y 594.419,Z 214.443,A -85,B 0,C 180,E1 -1252.526,E2 -1252.526} C_VEL
LIN {X 0,Y 594.389,Z 214.449,A -85,B 0,C 180,E1 -1255.251,E2 -1255.251} C_VEL
LIN {X 0,Y 594.394,Z 214.447,A -85,B 0,C 180,E1 -1257.966,E2 -1257.966} C_VEL
LIN {X 0,Y 594.422,Z 214.443,A -85,B 0,C 180,E1 -1260.676,E2 -1260.676} C_VEL
LIN {X 0,Y 594.378,Z 214.451,A -85,B 0,C 180,E1 -1263.388,E2 -1263.388} C_VEL
LIN {X 0,Y 594.366,Z 214.45,A -85,B 0,C 180,E1 -1266.108,E2 -1266.108} C_VEL
LIN {X 0,Y 594.398,Z 214.447,A -85,B 0,C 180,E1 -1268.841,E2 -1268.841} C_VEL
LIN {X 0,Y 594.369,Z 214.452,A -85,B 0,C 180,E1 -1271.595,E2 -1271.595} C_VEL
LIN {X 0,Y 594.303,Z 214.779,A -85,B 0,C 180,E1 -1272.368,E2 -1272.368} C_VEL
LIN {X 0,Y 594.286,Z 218.07,A -85,B 0,C 180,E1 -1275.079,E2 -1275.079} C_VEL
LIN {X 0,Y 594.276,Z 218.341,A -85,B 0,C 180,E1 -1275.305,E2 -1275.305} C_VEL
LIN {X 0,Y 593.605,Z 219.078,A -85,B 0,C 180,E1 -1275.866,E2 -1275.866} C_VEL
LIN {X 0,Y 590.747,Z 220.411,A -85,B 0,C 180,E1 -1276.775,E2 -1276.775} C_VEL
LIN {X 0,Y 588.334,Z 221.489,A -85,B 0,C 180,E1 -1277.507,E2 -1277.507} C_VEL
LIN {X 0,Y 587.299,Z 222.246,A -85,B 0,C 180,E1 -1278.072,E2 -1278.072} C_VEL
LIN {X 0,Y 587.215,Z 222.48,A -85,B 0,C 180,E1 -1278.264,E2 -1278.264} C_VEL
LIN {X 0,Y 587.164,Z 225.68,A -85,B 0,C 180,E1 -1281.042,E2 -1281.042} C_VEL
LIN {X 0,Y 587.164,Z 229.164,A -85,B 0,C 180,E1 -1284.012,E2 -1284.012} C_VEL
LIN {X 0,Y 587.101,Z 233.134,A -85,B 0,C 180,E1 -1287.056,E2 -1287.056} C_VEL
LIN {X 0,Y 587.14,Z 237.284,A -85,B 0,C 180,E1 -1290.179,E2 -1290.179} C_VEL
LIN {X 0,Y 587.104,Z 241.2,A -85,B 0,C 180,E1 -1293.078,E2 -1293.078} C_VEL
LIN {X 0,Y 587.118,Z 243.676,A -85,B 0,C 180,E1 -1294.892,E2 -1294.892} C_VEL
LIN {X 0,Y 587.734,Z 249.191,A -85,B 0,C 180,E1 -1295.026,E2 -1295.026} C_VEL
LIN {X 0,Y 587.656,Z 261.767,A -85,B 0,C 180,E1 -1295.378,E2 -1295.378} C_VEL
LIN {X 0,Y 587.549,Z 274.454,A -85,B 0,C 180,E1 -1295.88,E2 -1295.88} C_VEL
LIN {X 0,Y 587.439,Z 286.627,A -85,B 0,C 180,E1 -1296.525,E2 -1296.525} C_VEL
LIN {X 0,Y 587.383,Z 297.774,A -85,B 0,C 180,E1 -1297.279,E2 -1297.279} C_VEL
LIN {X 0,Y 587.321,Z 307.928,A -85,B 0,C 180,E1 -1298.132,E2 -1298.132} C_VEL
LIN {X 0,Y 587.274,Z 317.377,A -85,B 0,C 180,E1 -1299.123,E2 -1299.123} C_VEL
LIN {X 0,Y 587.229,Z 324.31,A -85,B 0,C 180,E1 -1300.009,E2 -1300.009} C_VEL
LIN {X 0,Y 587.195,Z 331.651,A -85,B 0,C 180,E1 -1301.167,E2 -1301.167} C_VEL
LIN {X 0,Y 587.207,Z 336.301,A -85,B 0,C 180,E1 -1302.095,E2 -1302.095} C_VEL
LIN {X 0,Y 587.17,Z 340.314,A -85,B 0,C 180,E1 -1303.104,E2 -1303.104} C_VEL
LIN {X 0,Y 587.161,Z 343.289,A -85,B 0,C 180,E1 -1304.097,E2 -1304.097} C_VEL
LIN {X 0,Y 587.171,Z 345.344,A -85,B 0,C 180,E1 -1305.075,E2 -1305.075} C_VEL
LIN {X 0,Y 587.122,Z 346.56,A -85,B 0,C 180,E1 -1306.031,E2 -1306.031} C_VEL
LIN {X 0,Y 587.154,Z 346.991,A -85,B 0,C 180,E1 -1306.98,E2 -1306.98} C_VEL
LIN {X 0,Y 587.146,Z 346.663,A -85,B 0,C 180,E1 -1307.91,E2 -1307.91} C_VEL
LIN {X 0,Y 587.116,Z 345.452,A -85,B 0,C 180,E1 -1308.947,E2 -1308.947} C_VEL
LIN {X 0,Y 587.145,Z 343.271,A -85,B 0,C 180,E1 -1309.999,E2 -1309.999} C_VEL
LIN {X 0,Y 587.175,Z 339.996,A -85,B 0,C 180,E1 -1311.075,E2 -1311.075} C_VEL
LIN {X 0,Y 587.174,Z 335.44,A -85,B 0,C 180,E1 -1312.179,E2 -1312.179} C_VEL
LIN {X 0,Y 587.22,Z 329.412,A -85,B 0,C 180,E1 -1313.306,E2 -1313.306} C_VEL
LIN {X 0,Y 587.235,Z 322.679,A -85,B 0,C 180,E1 -1314.309,E2 -1314.309} C_VEL
LIN {X 0,Y 587.317,Z 314.191,A -85,B 0,C 180,E1 -1315.325,E2 -1315.325} C_VEL
LIN {X 0,Y 587.357,Z 304.147,A -85,B 0,C 180,E1 -1316.297,E2 -1316.297} C_VEL
LIN {X 0,Y 587.439,Z 294.365,A -85,B 0,C 180,E1 -1317.062,E2 -1317.062} C_VEL
LIN {X 0,Y 587.484,Z 284.013,A -85,B 0,C 180,E1 -1317.718,E2 -1317.718} C_VEL
LIN {X 0,Y 587.576,Z 271.362,A -85,B 0,C 180,E1 -1318.347,E2 -1318.347} C_VEL
LIN {X 0,Y 587.682,Z 258.554,A -85,B 0,C 180,E1 -1318.817,E2 -1318.817} C_VEL
LIN {X 0,Y 587.609,Z 246.749,A -85,B 0,C 180,E1 -1319.119,E2 -1319.119} C_VEL
LIN {X 0,Y 587.138,Z 243.68,A -85,B 0,C 180,E1 -1319.195,E2 -1319.195} C_VEL
LIN {X 0,Y 587.132,Z 240.682,A -85,B 0,C 180,E1 -1321.393,E2 -1321.393} C_VEL
LIN {X 0,Y 587.149,Z 237.357,A -85,B 0,C 180,E1 -1323.857,E2 -1323.857} C_VEL
LIN {X 0,Y 587.169,Z 234.515,A -85,B 0,C 180,E1 -1325.987,E2 -1325.987} C_VEL
LIN {X 0,Y 587.132,Z 231.578,A -85,B 0,C 180,E1 -1328.219,E2 -1328.219} C_VEL
LIN {X 0,Y 587.188,Z 227.813,A -85,B 0,C 180,E1 -1331.146,E2 -1331.146} C_VEL
LIN {X 0,Y 587.19,Z 224.508,A -85,B 0,C 180,E1 -1334.022,E2 -1334.022} C_VEL
LIN {X 0,Y 587.18,Z 221.908,A -85,B 0,C 180,E1 -1336.15,E2 -1336.15} C_VEL
LIN {X 0,Y 587.269,Z 218.525,A -85,B 0,C 180,E1 -1338.962,E2 -1338.962} C_VEL
LIN {X 0,Y 587.237,Z 215.341,A -85,B 0,C 180,E1 -1341.743,E2 -1341.743} C_VEL
LIN {X 0,Y 587.309,Z 215.329,A -85,B 0,C 180,E1 -1343.818,E2 -1343.818} C_VEL
LIN {X 0,Y 587.313,Z 215.331,A -85,B 0,C 180,E1 -1345.883,E2 -1345.883} C_VEL
LIN {X 0,Y 587.357,Z 215.323,A -85,B 0,C 180,E1 -1347.943,E2 -1347.943} C_VEL
LIN {X 0,Y 587.39,Z 215.321,A -85,B 0,C 180,E1 -1350.686,E2 -1350.686} C_VEL
LIN {X 0,Y 587.325,Z 215.327,A -85,B 0,C 180,E1 -1353.43,E2 -1353.43} C_VEL
LIN {X 0,Y 587.355,Z 215.325,A -85,B 0,C 180,E1 -1355.493,E2 -1355.493} C_VEL
LIN {X 0,Y 587.359,Z 215.322,A -85,B 0,C 180,E1 -1358.256,E2 -1358.256} C_VEL
LIN {X 0,Y 587.365,Z 215.323,A -85,B 0,C 180,E1 -1361.151,E2 -1361.151} C_VEL
LIN {X 0,Y 587.35,Z 215.323,A -85,B 0,C 180,E1 -1364.262,E2 -1364.262} C_VEL
LIN {X 0,Y 587.35,Z 215.326,A -85,B 0,C 180,E1 -1367.406,E2 -1367.406} C_VEL
LIN {X 0,Y 587.325,Z 215.326,A -85,B 0,C 180,E1 -1370.305,E2 -1370.305} C_VEL
LIN {X 0,Y 587.353,Z 215.326,A -85,B 0,C 180,E1 -1373.258,E2 -1373.258} C_VEL
LIN {X 0,Y 587.354,Z 215.322,A -85,B 0,C 180,E1 -1376.278,E2 -1376.278} C_VEL
LIN {X 0,Y 587.342,Z 215.327,A -85,B 0,C 180,E1 -1379.136,E2 -1379.136} C_VEL
LIN {X 0,Y 587.349,Z 215.325,A -85,B 0,C 180,E1 -1381.84,E2 -1381.84} C_VEL
LIN {X 0,Y 587.347,Z 215.324,A -85,B 0,C 180,E1 -1384.351,E2 -1384.351} C_VEL
LIN {X 0,Y 587.339,Z 215.325,A -85,B 0,C 180,E1 -1386.748,E2 -1386.748} C_VEL
LIN {X 0,Y 587.337,Z 215.324,A -85,B 0,C 180,E1 -1389.36,E2 -1389.36} C_VEL
LIN {X 0,Y 587.326,Z 215.327,A -85,B 0,C 180,E1 -1392.109,E2 -1392.109} C_VEL
LIN {X 0,Y 587.306,Z 215.329,A -85,B 0,C 180,E1 -1395.09,E2 -1395.09} C_VEL
LIN {X 0,Y 587.344,Z 215.324,A -85,B 0,C 180,E1 -1397.929,E2 -1397.929} C_VEL
LIN {X 0,Y 587.328,Z 215.326,A -85,B 0,C 180,E1 -1401.059,E2 -1401.059} C_VEL
LIN {X 0,Y 587.348,Z 215.325,A -85,B 0,C 180,E1 -1403.293,E2 -1403.293} C_VEL
LIN {X 0,Y 587.361,Z 215.323,A -85,B 0,C 180,E1 -1405.782,E2 -1405.782} C_VEL
LIN {X 0,Y 587.347,Z 215.324,A -85,B 0,C 180,E1 -1408.233,E2 -1408.233} C_VEL
LIN {X 0,Y 587.347,Z 215.323,A -85,B 0,C 180,E1 -1410.867,E2 -1410.867} C_VEL
LIN {X 0,Y 587.353,Z 215.326,A -85,B 0,C 180,E1 -1413.821,E2 -1413.821} C_VEL
LIN {X 0,Y 587.336,Z 215.327,A -85,B 0,C 180,E1 -1415.995,E2 -1415.995} C_VEL
LIN {X 0,Y 587.324,Z 215.327,A -85,B 0,C 180,E1 -1418.227,E2 -1418.227} C_VEL
LIN {X 0,Y 587.347,Z 215.325,A -85,B 0,C 180,E1 -1421.153,E2 -1421.153} C_VEL
LIN {X 0,Y 587.354,Z 215.326,A -85,B 0,C 180,E1 -1423.313,E2 -1423.313} C_VEL
LIN {X 0,Y 587.356,Z 215.323,A -85,B 0,C 180,E1 -1426.156,E2 -1426.156} C_VEL
LIN {X 0,Y 587.344,Z 215.324,A -85,B 0,C 180,E1 -1428.964,E2 -1428.964} C_VEL
LIN {X 0,Y 587.326,Z 215.329,A -85,B 0,C 180,E1 -1431.745,E2 -1431.745} C_VEL
LIN {X 0,Y 587.332,Z 215.327,A -85,B 0,C 180,E1 -1433.819,E2 -1433.819} C_VEL
LIN {X 0,Y 587.315,Z 215.328,A -85,B 0,C 180,E1 -1435.884,E2 -1435.884} C_VEL
LIN {X 0,Y 587.357,Z 215.323,A -85,B 0,C 180,E1 -1437.944,E2 -1437.944} C_VEL
LIN {X 0,Y 587.383,Z 215.319,A -85,B 0,C 180,E1 -1440.687,E2 -1440.687} C_VEL
LIN {X 0,Y 587.33,Z 215.327,A -85,B 0,C 180,E1 -1443.431,E2 -1443.431} C_VEL
LIN {X 0,Y 587.363,Z 215.322,A -85,B 0,C 180,E1 -1445.494,E2 -1445.494} C_VEL
LIN {X 0,Y 587.344,Z 215.327,A -85,B 0,C 180,E1 -1448.257,E2 -1448.257} C_VEL
LIN {X 0,Y 587.353,Z 215.323,A -85,B 0,C 180,E1 -1451.135,E2 -1451.135} C_VEL
LIN {X 0,Y 587.361,Z 215.325,A -85,B 0,C 180,E1 -1454.258,E2 -1454.258} C_VEL
LIN {X 0,Y 587.362,Z 215.322,A -85,B 0,C 180,E1 -1457.407,E2 -1457.407} C_VEL
LIN {X 0,Y 587.331,Z 215.329,A -85,B 0,C 180,E1 -1460.306,E2 -1460.306} C_VEL
LIN {X 0,Y 587.323,Z 215.326,A -85,B 0,C 180,E1 -1463.26,E2 -1463.26} C_VEL
LIN {X 0,Y 587.34,Z 215.328,A -85,B 0,C 180,E1 -1466.279,E2 -1466.279} C_VEL
LIN {X 0,Y 587.355,Z 215.323,A -85,B 0,C 180,E1 -1469.134,E2 -1469.134} C_VEL
LIN {X 0,Y 587.347,Z 215.324,A -85,B 0,C 180,E1 -1471.836,E2 -1471.836} C_VEL
LIN {X 0,Y 587.349,Z 215.324,A -85,B 0,C 180,E1 -1474.347,E2 -1474.347} C_VEL
LIN {X 0,Y 587.349,Z 215.323,A -85,B 0,C 180,E1 -1477.608,E2 -1477.608} C_VEL
LIN {X 0,Y 587.314,Z 215.328,A -85,B 0,C 180,E1 -1480.255,E2 -1480.255} C_VEL
LIN {X 0,Y 587.318,Z 215.328,A -85,B 0,C 180,E1 -1483.118,E2 -1483.118} C_VEL
LIN {X 0,Y 587.317,Z 215.327,A -85,B 0,C 180,E1 -1486.049,E2 -1486.049} C_VEL
LIN {X 0,Y 587.34,Z 215.328,A -85,B 0,C 180,E1 -1488.925,E2 -1488.925} C_VEL
LIN {X 0,Y 587.327,Z 215.327,A -85,B 0,C 180,E1 -1491.52,E2 -1491.52} C_VEL
LIN {X 0,Y 587.349,Z 215.462,A -85,B 0,C 180,E1 -1493.733,E2 -1493.733} C_VEL
LIN {X 0,Y 587.666,Z 219.268,A -85,B 0,C 180,E1 -1494.967,E2 -1494.967} C_VEL
LIN {X 0,Y 587.654,Z 225.269,A -85,B 0,C 180,E1 -1496.842,E2 -1496.842} C_VEL
LIN {X 0,Y 587.54,Z 233.875,A -85,B 0,C 180,E1 -1499.457,E2 -1499.457} C_VEL
LIN {X 0,Y 587.508,Z 243.402,A -85,B 0,C 180,E1 -1502.279,E2 -1502.279} C_VEL
LIN {X 0,Y 587.447,Z 252.365,A -85,B 0,C 180,E1 -1504.868,E2 -1504.868} C_VEL
LIN {X 0,Y 587.381,Z 261.633,A -85,B 0,C 180,E1 -1507.488,E2 -1507.488} C_VEL
LIN {X 0,Y 587.345,Z 270.9,A -85,B 0,C 180,E1 -1510.061,E2 -1510.061} C_VEL
LIN {X 0,Y 587.292,Z 281.489,A -85,B 0,C 180,E1 -1512.95,E2 -1512.95} C_VEL
LIN {X 0,Y 587.253,Z 292.031,A -85,B 0,C 180,E1 -1515.784,E2 -1515.784} C_VEL
LIN {X 0,Y 587.203,Z 299.57,A -85,B 0,C 180,E1 -1517.789,E2 -1517.789} C_VEL
LIN {X 0,Y 587.729,Z 305.213,A -85,B 0,C 180,E1 -1517.899,E2 -1517.899} C_VEL
LIN {X 0,Y 587.684,Z 318.485,A -85,B 0,C 180,E1 -1518.226,E2 -1518.226} C_VEL
LIN {X 0,Y 587.566,Z 330.41,A -85,B 0,C 180,E1 -1518.656,E2 -1518.656} C_VEL
LIN {X 0,Y 587.479,Z 342.202,A -85,B 0,C 180,E1 -1519.226,E2 -1519.226} C_VEL
LIN {X 0,Y 587.467,Z 353.471,A -85,B 0,C 180,E1 -1519.923,E2 -1519.923} C_VEL
LIN {X 0,Y 587.385,Z 363.643,A -85,B 0,C 180,E1 -1520.704,E2 -1520.704} C_VEL
LIN {X 0,Y 587.331,Z 372.784,A -85,B 0,C 180,E1 -1521.571,E2 -1521.571} C_VEL
LIN {X 0,Y 587.259,Z 381.688,A -85,B 0,C 180,E1 -1522.608,E2 -1522.608} C_VEL
LIN {X 0,Y 587.195,Z 388.749,A -85,B 0,C 180,E1 -1523.628,E2 -1523.628} C_VEL
LIN {X 0,Y 587.211,Z 393.678,A -85,B 0,C 180,E1 -1524.505,E2 -1524.505} C_VEL
LIN {X 0,Y 587.189,Z 398.37,A -85,B 0,C 180,E1 -1525.538,E2 -1525.538} C_VEL
LIN {X 0,Y 587.193,Z 401.955,A -85,B 0,C 180,E1 -1526.569,E2 -1526.569} C_VEL
LIN {X 0,Y 587.132,Z 403.808,A -85,B 0,C 180,E1 -1527.255,E2 -1527.255} C_VEL
LIN {X 0,Y 587.141,Z 405.201,A -85,B 0,C 180,E1 -1527.942,E2 -1527.942} C_VEL
LIN {X 0,Y 587.14,Z 406.784,A -85,B 0,C 180,E1 -1529.314,E2 -1529.314} C_VEL
LIN {X 0,Y 587.137,Z 407,A -85,B 0,C 180,E1 -1530,E2 -1530} C_VEL
LIN {X 0,Y 587.147,Z 406.185,A -85,B 0,C 180,E1 -1531.371,E2 -1531.371} C_VEL
LIN {X 0,Y 587.141,Z 405.203,A -85,B 0,C 180,E1 -1532.058,E2 -1532.058} C_VEL
LIN {X 0,Y 587.132,Z 403.81,A -85,B 0,C 180,E1 -1532.744,E2 -1532.744} C_VEL
LIN {X 0,Y 587.213,Z 400.897,A -85,B 0,C 180,E1 -1533.774,E2 -1533.774} C_VEL
LIN {X 0,Y 587.147,Z 396.951,A -85,B 0,C 180,E1 -1534.806,E2 -1534.806} C_VEL
LIN {X 0,Y 587.218,Z 390.88,A -85,B 0,C 180,E1 -1536.011,E2 -1536.011} C_VEL
LIN {X 0,Y 587.245,Z 384.239,A -85,B 0,C 180,E1 -1537.046,E2 -1537.046} C_VEL
LIN {X 0,Y 587.299,Z 375.993,A -85,B 0,C 180,E1 -1538.083,E2 -1538.083} C_VEL
LIN {X 0,Y 587.343,Z 367.542,A -85,B 0,C 180,E1 -1538.949,E2 -1538.949} C_VEL
LIN {X 0,Y 587.421,Z 357.098,A -85,B 0,C 180,E1 -1539.816,E2 -1539.816} C_VEL
LIN {X 0,Y 587.475,Z 346.765,A -85,B 0,C 180,E1 -1540.511,E2 -1540.511} C_VEL
LIN {X 0,Y 587.53,Z 335.167,A -85,B 0,C 180,E1 -1541.133,E2 -1541.133} C_VEL
LIN {X 0,Y 587.624,Z 322.704,A -85,B 0,C 180,E1 -1541.636,E2 -1541.636} C_VEL
LIN {X 0,Y 587.715,Z 309.456,A -85,B 0,C 180,E1 -1542.013,E2 -1542.013} C_VEL
LIN {X 0,Y 587.545,Z 301.644,A -85,B 0,C 180,E1 -1542.17,E2 -1542.17} C_VEL
LIN {X 0,Y 587.201,Z 299.532,A -85,B 0,C 180,E1 -1542.221,E2 -1542.221} C_VEL
LIN {X 0,Y 587.257,Z 289.437,A -85,B 0,C 180,E1 -1544.91,E2 -1544.91} C_VEL
LIN {X 0,Y 587.303,Z 278.846,A -85,B 0,C 180,E1 -1547.767,E2 -1547.767} C_VEL
LIN {X 0,Y 587.377,Z 268.255,A -85,B 0,C 180,E1 -1550.669,E2 -1550.669} C_VEL
LIN {X 0,Y 587.434,Z 257.664,A -85,B 0,C 180,E1 -1553.627,E2 -1553.627} C_VEL
LIN {X 0,Y 587.486,Z 248.397,A -85,B 0,C 180,E1 -1556.271,E2 -1556.271} C_VEL
LIN {X 0,Y 587.476,Z 240.453,A -85,B 0,C 180,E1 -1558.588,E2 -1558.588} C_VEL
LIN {X 0,Y 587.566,Z 232.51,A -85,B 0,C 180,E1 -1560.952,E2 -1560.952} C_VEL
LIN {X 0,Y 587.672,Z 223.243,A -85,B 0,C 180,E1 -1563.786,E2 -1563.786} C_VEL
LIN {X 0,Y 587.591,Z 216.623,A -85,B 0,C 180,E1 -1565.878,E2 -1565.878} C_VEL
LIN {X 0,Y 587.314,Z 215.331,A -85,B 0,C 180,E1 -1566.322,E2 -1566.322} C_VEL
LIN {X 0,Y 587.318,Z 215.329,A -85,B 0,C 180,E1 -1568.939,E2 -1568.939} C_VEL
LIN {X 0,Y 587.339,Z 215.326,A -85,B 0,C 180,E1 -1572.073,E2 -1572.073} C_VEL
LIN {X 0,Y 587.317,Z 215.328,A -85,B 0,C 180,E1 -1575.088,E2 -1575.088} C_VEL
LIN {X 0,Y 587.354,Z 215.324,A -85,B 0,C 180,E1 -1577.927,E2 -1577.927} C_VEL
LIN {X 0,Y 587.336,Z 215.326,A -85,B 0,C 180,E1 -1581.057,E2 -1581.057} C_VEL
LIN {X 0,Y 587.349,Z 215.324,A -85,B 0,C 180,E1 -1583.291,E2 -1583.291} C_VEL
LIN {X 0,Y 587.363,Z 215.324,A -85,B 0,C 180,E1 -1585.779,E2 -1585.779} C_VEL
LIN {X 0,Y 587.343,Z 215.326,A -85,B 0,C 180,E1 -1588.23,E2 -1588.23} C_VEL
LIN {X 0,Y 587.35,Z 215.324,A -85,B 0,C 180,E1 -1590.865,E2 -1590.865} C_VEL
LIN {X 0,Y 587.362,Z 215.322,A -85,B 0,C 180,E1 -1593.817,E2 -1593.817} C_VEL
LIN {X 0,Y 587.335,Z 215.326,A -85,B 0,C 180,E1 -1595.993,E2 -1595.993} C_VEL
LIN {X 0,Y 587.348,Z 215.324,A -85,B 0,C 180,E1 -1598.962,E2 -1598.962} C_VEL
LIN {X 0,Y 587.351,Z 215.324,A -85,B 0,C 180,E1 -1601.15,E2 -1601.15} C_VEL
LIN {X 0,Y 587.325,Z 215.327,A -85,B 0,C 180,E1 -1604.024,E2 -1604.024} C_VEL
LIN {X 0,Y 587.36,Z 215.323,A -85,B 0,C 180,E1 -1606.153,E2 -1606.153} C_VEL
LIN {X 0,Y 587.336,Z 215.327,A -85,B 0,C 180,E1 -1608.961,E2 -1608.961} C_VEL
LIN {X 0,Y 587.365,Z 215.323,A -85,B 0,C 180,E1 -1611.744,E2 -1611.744} C_VEL
LIN {X 0,Y 587.363,Z 215.322,A -85,B 0,C 180,E1 -1614.506,E2 -1614.506} C_VEL
LIN {X 0,Y 587.373,Z 215.323,A -85,B 0,C 180,E1 -1617.256,E2 -1617.256} C_VEL
LIN {X 0,Y 587.376,Z 215.321,A -85,B 0,C 180,E1 -1619.999,E2 -1619.999} C_VEL
LIN {X 0,Y 587.374,Z 215.321,A -85,B 0,C 180,E1 -1622.742,E2 -1622.742} C_VEL
LIN {X 0,Y 587.353,Z 215.326,A -85,B 0,C 180,E1 -1625.492,E2 -1625.492} C_VEL
LIN {X 0,Y 587.37,Z 215.322,A -85,B 0,C 180,E1 -1628.254,E2 -1628.254} C_VEL
LIN {X 0,Y 587.341,Z 215.326,A -85,B 0,C 180,E1 -1631.132,E2 -1631.132} C_VEL
LIN {X 0,Y 587.246,Z 215.535,A -85,B 0,C 180,E1 -1632.439,E2 -1632.439} C_VEL
LIN {X 0,Y 587.232,Z 218.981,A -85,B 0,C 180,E1 -1635.293,E2 -1635.293} C_VEL
LIN {X 0,Y 587.221,Z 221.472,A -85,B 0,C 180,E1 -1637.408,E2 -1637.408} C_VEL
LIN {X 0,Y 587.215,Z 222.48,A -85,B 0,C 180,E1 -1638.264,E2 -1638.264} C_VEL
LIN {X 0,Y 586.542,Z 223.217,A -85,B 0,C 180,E1 -1638.831,E2 -1638.831} C_VEL
LIN {X 0,Y 583.655,Z 224.561,A -85,B 0,C 180,E1 -1639.75,E2 -1639.75} C_VEL
LIN {X 0,Y 581.215,Z 225.615,A -85,B 0,C 180,E1 -1640.49,E2 -1640.49} C_VEL
LIN {X 0,Y 580.167,Z 226.335,A -85,B 0,C 180,E1 -1641.062,E2 -1641.062} C_VEL
LIN {X 0,Y 580.082,Z 226.555,A -85,B 0,C 180,E1 -1641.256,E2 -1641.256} C_VEL
LIN {X 0,Y 580.103,Z 229.991,A -85,B 0,C 180,E1 -1644.323,E2 -1644.323} C_VEL
LIN {X 0,Y 580.022,Z 233.931,A -85,B 0,C 180,E1 -1647.414,E2 -1647.414} C_VEL
LIN {X 0,Y 580.026,Z 237.046,A -85,B 0,C 180,E1 -1649.786,E2 -1649.786} C_VEL
LIN {X 0,Y 580.013,Z 240.28,A -85,B 0,C 180,E1 -1652.216,E2 -1652.216} C_VEL
LIN {X 0,Y 580.031,Z 243.673,A -85,B 0,C 180,E1 -1654.738,E2 -1654.738} C_VEL
LIN {X 0,Y 580.804,Z 249.865,A -85,B 0,C 180,E1 -1654.897,E2 -1654.897} C_VEL
LIN {X 0,Y 580.696,Z 262.111,A -85,B 0,C 180,E1 -1655.248,E2 -1655.248} C_VEL
LIN {X 0,Y 580.595,Z 274.164,A -85,B 0,C 180,E1 -1655.731,E2 -1655.731} C_VEL
LIN {X 0,Y 580.488,Z 285.114,A -85,B 0,C 180,E1 -1656.304,E2 -1656.304} C_VEL
LIN {X 0,Y 580.41,Z 296.631,A -85,B 0,C 180,E1 -1657.074,E2 -1657.074} C_VEL
LIN {X 0,Y 580.341,Z 306.409,A -85,B 0,C 180,E1 -1657.885,E2 -1657.885} C_VEL
LIN {X 0,Y 580.243,Z 315.558,A -85,B 0,C 180,E1 -1658.813,E2 -1658.813} C_VEL
LIN {X 0,Y 580.178,Z 322.986,A -85,B 0,C 180,E1 -1659.736,E2 -1659.736} C_VEL
LIN {X 0,Y 580.114,Z 330.282,A -85,B 0,C 180,E1 -1660.857,E2 -1660.857} C_VEL
LIN {X 0,Y 580.107,Z 336.45,A -85,B 0,C 180,E1 -1662.066,E2 -1662.066} C_VEL
LIN {X 0,Y 580.082,Z 340.276,A -85,B 0,C 180,E1 -1663.045,E2 -1663.045} C_VEL
LIN {X 0,Y 580.063,Z 342.274,A -85,B 0,C 180,E1 -1663.676,E2 -1663.676} C_VEL
LIN {X 0,Y 580.071,Z 344.599,A -85,B 0,C 180,E1 -1664.643,E2 -1664.643} C_VEL
LIN {X 0,Y 580.056,Z 346.154,A -85,B 0,C 180,E1 -1665.628,E2 -1665.628} C_VEL
LIN {X 0,Y 580.02,Z 346.913,A -85,B 0,C 180,E1 -1666.634,E2 -1666.634} C_VEL
LIN {X 0,Y 580.049,Z 346.844,A -85,B 0,C 180,E1 -1667.651,E2 -1667.651} C_VEL
LIN {X 0,Y 580.027,Z 345.882,A -85,B 0,C 180,E1 -1668.695,E2 -1668.695} C_VEL
LIN {X 0,Y 580.052,Z 343.239,A -85,B 0,C 180,E1 -1670.048,E2 -1670.048} C_VEL
LIN {X 0,Y 580.094,Z 340.61,A -85,B 0,C 180,E1 -1670.951,E2 -1670.951} C_VEL
LIN {X 0,Y 580.09,Z 336.785,A -85,B 0,C 180,E1 -1671.949,E2 -1671.949} C_VEL
LIN {X 0,Y 580.119,Z 331.129,A -85,B 0,C 180,E1 -1673.086,E2 -1673.086} C_VEL
LIN {X 0,Y 580.165,Z 323.713,A -85,B 0,C 180,E1 -1674.252,E2 -1674.252} C_VEL
LIN {X 0,Y 580.24,Z 315.349,A -85,B 0,C 180,E1 -1675.301,E2 -1675.301} C_VEL
LIN {X 0,Y 580.305,Z 307.079,A -85,B 0,C 180,E1 -1676.145,E2 -1676.145} C_VEL
LIN {X 0,Y 580.386,Z 297.091,A -85,B 0,C 180,E1 -1676.982,E2 -1676.982} C_VEL
LIN {X 0,Y 580.503,Z 286.336,A -85,B 0,C 180,E1 -1677.71,E2 -1677.71} C_VEL
LIN {X 0,Y 580.61,Z 274.793,A -85,B 0,C 180,E1 -1678.33,E2 -1678.33} C_VEL
LIN {X 0,Y 580.723,Z 262.121,A -85,B 0,C 180,E1 -1678.841,E2 -1678.841} C_VEL
LIN {X 0,Y 580.784,Z 248.832,A -85,B 0,C 180,E1 -1679.219,E2 -1679.219} C_VEL
LIN {X 0,Y 580.047,Z 243.686,A -85,B 0,C 180,E1 -1679.341,E2 -1679.341} C_VEL
LIN {X 0,Y 580.042,Z 239.862,A -85,B 0,C 180,E1 -1682.185,E2 -1682.185} C_VEL
LIN {X 0,Y 580.062,Z 236.245,A -85,B 0,C 180,E1 -1684.909,E2 -1684.909} C_VEL
LIN {X 0,Y 580.092,Z 233.259,A -85,B 0,C 180,E1 -1687.19,E2 -1687.19} C_VEL
LIN {X 0,Y 580.063,Z 229.54,A -85,B 0,C 180,E1 -1690.17,E2 -1690.17} C_VEL
LIN {X 0,Y 580.122,Z 226.136,A -85,B 0,C 180,E1 -1693.142,E2 -1693.142} C_VEL
LIN {X 0,Y 580.135,Z 222.691,A -85,B 0,C 180,E1 -1695.979,E2 -1695.979} C_VEL
LIN {X 0,Y 580.193,Z 219.278,A -85,B 0,C 180,E1 -1698.853,E2 -1698.853} C_VEL
LIN {X 0,Y 580.178,Z 216.83,A -85,B 0,C 180,E1 -1700.94,E2 -1700.94} C_VEL
LIN {X 0,Y 580.182,Z 216.219,A -85,B 0,C 180,E1 -1701.642,E2 -1701.642} C_VEL
LIN {X 0,Y 580.268,Z 216.206,A -85,B 0,C 180,E1 -1703.742,E2 -1703.742} C_VEL
LIN {X 0,Y 580.269,Z 216.209,A -85,B 0,C 180,E1 -1705.833,E2 -1705.833} C_VEL
LIN {X 0,Y 580.327,Z 216.199,A -85,B 0,C 180,E1 -1707.918,E2 -1707.918} C_VEL
LIN {X 0,Y 580.359,Z 216.197,A -85,B 0,C 180,E1 -1710.694,E2 -1710.694} C_VEL
LIN {X 0,Y 580.276,Z 216.204,A -85,B 0,C 180,E1 -1713.472,E2 -1713.472} C_VEL
LIN {X 0,Y 580.319,Z 216.201,A -85,B 0,C 180,E1 -1715.56,E2 -1715.56} C_VEL
LIN {X 0,Y 580.322,Z 216.198,A -85,B 0,C 180,E1 -1718.357,E2 -1718.357} C_VEL
LIN {X 0,Y 580.317,Z 216.201,A -85,B 0,C 180,E1 -1721.209,E2 -1721.209} C_VEL
LIN {X 0,Y 580.312,Z 216.201,A -85,B 0,C 180,E1 -1724.018,E2 -1724.018} C_VEL
LIN {X 0,Y 580.305,Z 216.201,A -85,B 0,C 180,E1 -1726.918,E2 -1726.918} C_VEL
LIN {X 0,Y 580.297,Z 216.204,A -85,B 0,C 180,E1 -1729.823,E2 -1729.823} C_VEL
LIN {X 0,Y 580.316,Z 216.199,A -85,B 0,C 180,E1 -1732.802,E2 -1732.802} C_VEL
LIN {X 0,Y 580.289,Z 216.204,A -85,B 0,C 180,E1 -1735.849,E2 -1735.849} C_VEL
LIN {X 0,Y 580.293,Z 216.205,A -85,B 0,C 180,E1 -1738.186,E2 -1738.186} C_VEL
LIN {X 0,Y 580.279,Z 216.205,A -85,B 0,C 180,E1 -1740.697,E2 -1740.697} C_VEL
LIN {X 0,Y 580.293,Z 216.202,A -85,B 0,C 180,E1 -1743.318,E2 -1743.318} C_VEL
LIN {X 0,Y 580.309,Z 216.2,A -85,B 0,C 180,E1 -1745.768,E2 -1745.768} C_VEL
LIN {X 0,Y 580.28,Z 216.204,A -85,B 0,C 180,E1 -1748.147,E2 -1748.147} C_VEL
LIN {X 0,Y 580.31,Z 216.201,A -85,B 0,C 180,E1 -1750.843,E2 -1750.843} C_VEL
LIN {X 0,Y 580.28,Z 216.206,A -85,B 0,C 180,E1 -1753.658,E2 -1753.658} C_VEL
LIN {X 0,Y 580.277,Z 216.204,A -85,B 0,C 180,E1 -1756.61,E2 -1756.61} C_VEL
LIN {X 0,Y 580.295,Z 216.203,A -85,B 0,C 180,E1 -1759.159,E2 -1759.159} C_VEL
LIN {X 0,Y 580.285,Z 216.207,A -85,B 0,C 180,E1 -1761.928,E2 -1761.928} C_VEL
LIN {X 0,Y 580.282,Z 216.205,A -85,B 0,C 180,E1 -1764.457,E2 -1764.457} C_VEL
LIN {X 0,Y 580.286,Z 216.203,A -85,B 0,C 180,E1 -1766.977,E2 -1766.977} C_VEL
LIN {X 0,Y 580.305,Z 216.201,A -85,B 0,C 180,E1 -1769.428,E2 -1769.428} C_VEL
LIN {X 0,Y 580.316,Z 216.199,A -85,B 0,C 180,E1 -1772.138,E2 -1772.138} C_VEL
LIN {X 0,Y 580.318,Z 216.2,A -85,B 0,C 180,E1 -1775.271,E2 -1775.271} C_VEL
LIN {X 0,Y 580.273,Z 216.205,A -85,B 0,C 180,E1 -1777.949,E2 -1777.949} C_VEL
LIN {X 0,Y 580.317,Z 216.202,A -85,B 0,C 180,E1 -1780.916,E2 -1780.916} C_VEL
LIN {X 0,Y 580.281,Z 216.204,A -85,B 0,C 180,E1 -1783.827,E2 -1783.827} C_VEL
LIN {X 0,Y 580.323,Z 216.2,A -85,B 0,C 180,E1 -1785.984,E2 -1785.984} C_VEL
LIN {X 0,Y 580.305,Z 216.201,A -85,B 0,C 180,E1 -1788.828,E2 -1788.828} C_VEL
LIN {X 0,Y 580.299,Z 216.205,A -85,B 0,C 180,E1 -1791.645,E2 -1791.645} C_VEL
LIN {X 0,Y 580.29,Z 216.203,A -85,B 0,C 180,E1 -1793.744,E2 -1793.744} C_VEL
LIN {X 0,Y 580.271,Z 216.205,A -85,B 0,C 180,E1 -1795.834,E2 -1795.834} C_VEL
LIN {X 0,Y 580.329,Z 216.199,A -85,B 0,C 180,E1 -1797.919,E2 -1797.919} C_VEL
LIN {X 0,Y 580.355,Z 216.194,A -85,B 0,C 180,E1 -1800.695,E2 -1800.695} C_VEL
LIN {X 0,Y 580.281,Z 216.206,A -85,B 0,C 180,E1 -1803.473,E2 -1803.473} C_VEL
LIN {X 0,Y 580.327,Z 216.198,A -85,B 0,C 180,E1 -1805.561,E2 -1805.561} C_VEL
LIN {X 0,Y 580.314,Z 216.203,A -85,B 0,C 180,E1 -1808.357,E2 -1808.357} C_VEL
LIN {X 0,Y 580.305,Z 216.201,A -85,B 0,C 180,E1 -1811.192,E2 -1811.192} C_VEL
LIN {X 0,Y 580.322,Z 216.199,A -85,B 0,C 180,E1 -1814.018,E2 -1814.018} C_VEL
LIN {X 0,Y 580.318,Z 216.201,A -85,B 0,C 180,E1 -1816.915,E2 -1816.915} C_VEL
LIN {X 0,Y 580.291,Z 216.203,A -85,B 0,C 180,E1 -1819.824,E2 -1819.824} C_VEL
LIN {X 0,Y 580.273,Z 216.204,A -85,B 0,C 180,E1 -1822.054,E2 -1822.054} C_VEL
LIN {X 0,Y 580.288,Z 216.206,A -85,B 0,C 180,E1 -1825.081,E2 -1825.081} C_VEL
LIN {X 0,Y 580.302,Z 216.201,A -85,B 0,C 180,E1 -1827.859,E2 -1827.859} C_VEL
LIN {X 0,Y 580.277,Z 216.205,A -85,B 0,C 180,E1 -1830.693,E2 -1830.693} C_VEL
LIN {X 0,Y 580.289,Z 216.206,A -85,B 0,C 180,E1 -1833.314,E2 -1833.314} C_VEL
LIN {X 0,Y 580.252,Z 216.211,A -85,B 0,C 180,E1 -1835.757,E2 -1835.757} C_VEL
LIN {X 0,Y 580.294,Z 216.206,A -85,B 0,C 180,E1 -1838.147,E2 -1838.147} C_VEL
LIN {X 0,Y 580.301,Z 216.202,A -85,B 0,C 180,E1 -1840.844,E2 -1840.844} C_VEL
LIN {X 0,Y 580.284,Z 216.203,A -85,B 0,C 180,E1 -1843.658,E2 -1843.658} C_VEL
LIN {X 0,Y 580.28,Z 216.206,A -85,B 0,C 180,E1 -1846.61,E2 -1846.61} C_VEL
LIN {X 0,Y 580.303,Z 216.203,A -85,B 0,C 180,E1 -1849.157,E2 -1849.157} C_VEL
LIN {X 0,Y 580.291,Z 216.203,A -85,B 0,C 180,E1 -1851.928,E2 -1851.928} C_VEL
LIN {X 0,Y 580.308,Z 216.329,A -85,B 0,C 180,E1 -1853.504,E2 -1853.504} C_VEL
LIN {X 0,Y 580.732,Z 220.592,A -85,B 0,C 180,E1 -1854.911,E2 -1854.911} C_VEL
LIN {X 0,Y 580.635,Z 228.535,A -85,B 0,C 180,E1 -1857.409,E2 -1857.409} C_VEL
LIN {X 0,Y 580.576,Z 237.803,A -85,B 0,C 180,E1 -1860.243,E2 -1860.243} C_VEL
LIN {X 0,Y 580.439,Z 247.07,A -85,B 0,C 180,E1 -1862.996,E2 -1862.996} C_VEL
LIN {X 0,Y 580.395,Z 256.337,A -85,B 0,C 180,E1 -1865.688,E2 -1865.688} C_VEL
LIN {X 0,Y 580.36,Z 265.604,A -85,B 0,C 180,E1 -1868.324,E2 -1868.324} C_VEL
LIN {X 0,Y 580.26,Z 276.195,A -85,B 0,C 180,E1 -1871.279,E2 -1871.279} C_VEL
LIN {X 0,Y 580.218,Z 285.463,A -85,B 0,C 180,E1 -1873.824,E2 -1873.824} C_VEL
LIN {X 0,Y 580.182,Z 296.054,A -85,B 0,C 180,E1 -1876.693,E2 -1876.693} C_VEL
LIN {X 0,Y 580.126,Z 299.529,A -85,B 0,C 180,E1 -1877.627,E2 -1877.627} C_VEL
LIN {X 0,Y 580.805,Z 305.213,A -85,B 0,C 180,E1 -1877.752,E2 -1877.752} C_VEL
LIN {X 0,Y 580.72,Z 318.485,A -85,B 0,C 180,E1 -1878.083,E2 -1878.083} C_VEL
LIN {X 0,Y 580.6,Z 330.626,A -85,B 0,C 180,E1 -1878.528,E2 -1878.528} C_VEL
LIN {X 0,Y 580.489,Z 342.203,A -85,B 0,C 180,E1 -1879.095,E2 -1879.095} C_VEL
LIN {X 0,Y 580.467,Z 353.472,A -85,B 0,C 180,E1 -1879.8,E2 -1879.8} C_VEL
LIN {X 0,Y 580.353,Z 363.643,A -85,B 0,C 180,E1 -1880.591,E2 -1880.591} C_VEL
LIN {X 0,Y 580.27,Z 372.784,A -85,B 0,C 180,E1 -1881.467,E2 -1881.467} C_VEL
LIN {X 0,Y 580.2,Z 381.688,A -85,B 0,C 180,E1 -1882.518,E2 -1882.518} C_VEL
LIN {X 0,Y 580.12,Z 388.469,A -85,B 0,C 180,E1 -1883.505,E2 -1883.505} C_VEL
LIN {X 0,Y 580.139,Z 393.678,A -85,B 0,C 180,E1 -1884.438,E2 -1884.438} C_VEL
LIN {X 0,Y 580.108,Z 398.37,A -85,B 0,C 180,E1 -1885.483,E2 -1885.483} C_VEL
LIN {X 0,Y 580.123,Z 401.955,A -85,B 0,C 180,E1 -1886.527,E2 -1886.527} C_VEL
LIN {X 0,Y 580.043,Z 403.808,A -85,B 0,C 180,E1 -1887.222,E2 -1887.222} C_VEL
LIN {X 0,Y 580.04,Z 405.201,A -85,B 0,C 180,E1 -1887.917,E2 -1887.917} C_VEL
LIN {X 0,Y 580.04,Z 406.784,A -85,B 0,C 180,E1 -1889.305,E2 -1889.305} C_VEL
LIN {X 0,Y 580.037,Z 407,A -85,B 0,C 180,E1 -1890,E2 -1890} C_VEL
LIN {X 0,Y 580.047,Z 406.185,A -85,B 0,C 180,E1 -1891.388,E2 -1891.388} C_VEL
LIN {X 0,Y 580.04,Z 405.202,A -85,B 0,C 180,E1 -1892.083,E2 -1892.083} C_VEL
LIN {X 0,Y 580.043,Z 403.81,A -85,B 0,C 180,E1 -1892.778,E2 -1892.778} C_VEL
LIN {X 0,Y 580.11,Z 400.897,A -85,B 0,C 180,E1 -1893.82,E2 -1893.82} C_VEL
LIN {X 0,Y 580.053,Z 396.951,A -85,B 0,C 180,E1 -1894.865,E2 -1894.865} C_VEL
LIN {X 0,Y 580.139,Z 390.88,A -85,B 0,C 180,E1 -1896.084,E2 -1896.084} C_VEL
LIN {X 0,Y 580.184,Z 384.239,A -85,B 0,C 180,E1 -1897.132,E2 -1897.132} C_VEL
LIN {X 0,Y 580.25,Z 375.993,A -85,B 0,C 180,E1 -1898.181,E2 -1898.181} C_VEL
LIN {X 0,Y 580.308,Z 367.542,A -85,B 0,C 180,E1 -1899.058,E2 -1899.058} C_VEL
LIN {X 0,Y 580.423,Z 357.099,A -85,B 0,C 180,E1 -1899.935,E2 -1899.935} C_VEL
LIN {X 0,Y 580.477,Z 346.766,A -85,B 0,C 180,E1 -1900.639,E2 -1900.639} C_VEL
LIN {X 0,Y 580.563,Z 335.603,A -85,B 0,C 180,E1 -1901.247,E2 -1901.247} C_VEL
LIN {X 0,Y 580.663,Z 323.78,A -85,B 0,C 180,E1 -1901.74,E2 -1901.74} C_VEL
LIN {X 0,Y 580.773,Z 310.37,A -85,B 0,C 180,E1 -1902.137,E2 -1902.137} C_VEL
LIN {X 0,Y 580.6,Z 302.359,A -85,B 0,C 180,E1 -1902.307,E2 -1902.307} C_VEL
LIN {X 0,Y 580.125,Z 299.532,A -85,B 0,C 180,E1 -1902.373,E2 -1902.373} C_VEL
LIN {X 0,Y 580.218,Z 289.437,A -85,B 0,C 180,E1 -1905.095,E2 -1905.095} C_VEL
LIN {X 0,Y 580.253,Z 278.846,A -85,B 0,C 180,E1 -1907.99,E2 -1907.99} C_VEL
LIN {X 0,Y 580.334,Z 268.493,A -85,B 0,C 180,E1 -1910.864,E2 -1910.864} C_VEL
LIN {X 0,Y 580.405,Z 258.988,A -85,B 0,C 180,E1 -1913.552,E2 -1913.552} C_VEL
LIN {X 0,Y 580.481,Z 249.223,A -85,B 0,C 180,E1 -1916.371,E2 -1916.371} C_VEL
LIN {X 0,Y 580.501,Z 240.453,A -85,B 0,C 180,E1 -1918.964,E2 -1918.964} C_VEL
LIN {X 0,Y 580.637,Z 231.347,A -85,B 0,C 180,E1 -1921.72,E2 -1921.72} C_VEL
LIN {X 0,Y 580.709,Z 223.323,A -85,B 0,C 180,E1 -1924.221,E2 -1924.221} C_VEL
LIN {X 0,Y 580.672,Z 218.351,A -85,B 0,C 180,E1 -1925.814,E2 -1925.814} C_VEL
LIN {X 0,Y 580.305,Z 216.204,A -85,B 0,C 180,E1 -1926.59,E2 -1926.59} C_VEL
LIN {X 0,Y 580.293,Z 216.205,A -85,B 0,C 180,E1 -1929.184,E2 -1929.184} C_VEL
LIN {X 0,Y 580.291,Z 216.204,A -85,B 0,C 180,E1 -1931.767,E2 -1931.767} C_VEL
LIN {X 0,Y 580.267,Z 216.208,A -85,B 0,C 180,E1 -1934.625,E2 -1934.625} C_VEL
LIN {X 0,Y 580.287,Z 216.206,A -85,B 0,C 180,E1 -1937.627,E2 -1937.627} C_VEL
LIN {X 0,Y 580.295,Z 216.203,A -85,B 0,C 180,E1 -1940.066,E2 -1940.066} C_VEL
LIN {X 0,Y 580.299,Z 216.203,A -85,B 0,C 180,E1 -1943.065,E2 -1943.065} C_VEL
LIN {X 0,Y 580.316,Z 216.202,A -85,B 0,C 180,E1 -1946.144,E2 -1946.144} C_VEL
LIN {X 0,Y 580.28,Z 216.205,A -85,B 0,C 180,E1 -1948.614,E2 -1948.614} C_VEL
LIN {X 0,Y 580.293,Z 216.204,A -85,B 0,C 180,E1 -1951.023,E2 -1951.023} C_VEL
LIN {X 0,Y 580.328,Z 216.199,A -85,B 0,C 180,E1 -1953.657,E2 -1953.657} C_VEL
LIN {X 0,Y 580.278,Z 216.207,A -85,B 0,C 180,E1 -1956.441,E2 -1956.441} C_VEL
LIN {X 0,Y 580.282,Z 216.207,A -85,B 0,C 180,E1 -1959.437,E2 -1959.437} C_VEL
LIN {X 0,Y 580.268,Z 216.208,A -85,B 0,C 180,E1 -1961.644,E2 -1961.644} C_VEL
LIN {X 0,Y 580.28,Z 216.206,A -85,B 0,C 180,E1 -1963.825,E2 -1963.825} C_VEL
LIN {X 0,Y 580.325,Z 216.2,A -85,B 0,C 180,E1 -1965.982,E2 -1965.982} C_VEL
LIN {X 0,Y 580.302,Z 216.204,A -85,B 0,C 180,E1 -1968.826,E2 -1968.826} C_VEL
LIN {X 0,Y 580.328,Z 216.199,A -85,B 0,C 180,E1 -1971.643,E2 -1971.643} C_VEL
LIN {X 0,Y 580.329,Z 216.199,A -85,B 0,C 180,E1 -1974.439,E2 -1974.439} C_VEL
LIN {X 0,Y 580.339,Z 216.2,A -85,B 0,C 180,E1 -1977.222,E2 -1977.222} C_VEL
LIN {X 0,Y 580.346,Z 216.197,A -85,B 0,C 180,E1 -1979.999,E2 -1979.999} C_VEL
LIN {X 0,Y 580.339,Z 216.197,A -85,B 0,C 180,E1 -1982.775,E2 -1982.775} C_VEL
LIN {X 0,Y 580.319,Z 216.202,A -85,B 0,C 180,E1 -1985.559,E2 -1985.559} C_VEL
LIN {X 0,Y 580.333,Z 216.199,A -85,B 0,C 180,E1 -1988.355,E2 -1988.355} C_VEL
LIN {X 0,Y 580.293,Z 216.204,A -85,B 0,C 180,E1 -1991.19,E2 -1991.19} C_VEL
LIN {X 0,Y 580.169,Z 216.399,A -85,B 0,C 180,E1 -1992.593,E2 -1992.593} C_VEL
LIN {X 0,Y 580.157,Z 218.968,A -85,B 0,C 180,E1 -1994.736,E2 -1994.736} C_VEL
LIN {X 0,Y 580.172,Z 221.515,A -85,B 0,C 180,E1 -1996.9,E2 -1996.9} C_VEL
LIN {X 0,Y 580.133,Z 224.953,A -85,B 0,C 180,E1 -1999.827,E2 -1999.827} C_VEL
LIN {X 0,Y 580.082,Z 226.555,A -85,B 0,C 180,E1 -2001.256,E2 -2001.256} C_VEL
LIN {X 0,Y 579.41,Z 227.248,A -85,B 0,C 180,E1 -2001.832,E2 -2001.832} C_VEL
LIN {X 0,Y 576.535,Z 228.536,A -85,B 0,C 180,E1 -2002.764,E2 -2002.764} C_VEL
LIN {X 0,Y 574.108,Z 229.583,A -85,B 0,C 180,E1 -2003.514,E2 -2003.514} C_VEL
LIN {X 0,Y 573.07,Z 230.323,A -85,B 0,C 180,E1 -2004.093,E2 -2004.093} C_VEL
LIN {X 0,Y 572.988,Z 230.552,A -85,B 0,C 180,E1 -2004.29,E2 -2004.29} C_VEL
LIN {X 0,Y 572.924,Z 233.713,A -85,B 0,C 180,E1 -2006.991,E2 -2006.991} C_VEL
LIN {X 0,Y 572.947,Z 236.877,A -85,B 0,C 180,E1 -2009.436,E2 -2009.436} C_VEL
LIN {X 0,Y 572.932,Z 240.478,A -85,B 0,C 180,E1 -2012.179,E2 -2012.179} C_VEL
LIN {X 0,Y 572.96,Z 243.713,A -85,B 0,C 180,E1 -2014.597,E2 -2014.597} C_VEL
LIN {X 0,Y 573.84,Z 250.717,A -85,B 0,C 180,E1 -2014.768,E2 -2014.768} C_VEL
LIN {X 0,Y 573.722,Z 263.467,A -85,B 0,C 180,E1 -2015.15,E2 -2015.15} C_VEL
LIN {X 0,Y 573.588,Z 275.281,A -85,B 0,C 180,E1 -2015.643,E2 -2015.643} C_VEL
LIN {X 0,Y 573.464,Z 286.359,A -85,B 0,C 180,E1 -2016.249,E2 -2016.249} C_VEL
LIN {X 0,Y 573.369,Z 297.909,A -85,B 0,C 180,E1 -2017.048,E2 -2017.048} C_VEL
LIN {X 0,Y 573.252,Z 308.103,A -85,B 0,C 180,E1 -2017.929,E2 -2017.929} C_VEL
LIN {X 0,Y 573.184,Z 316.994,A -85,B 0,C 180,E1 -2018.881,E2 -2018.881} C_VEL
LIN {X 0,Y 573.093,Z 324.324,A -85,B 0,C 180,E1 -2019.836,E2 -2019.836} C_VEL
LIN {X 0,Y 573.031,Z 331.563,A -85,B 0,C 180,E1 -2021.005,E2 -2021.005} C_VEL
LIN {X 0,Y 573.029,Z 336.281,A -85,B 0,C 180,E1 -2021.968,E2 -2021.968} C_VEL
LIN {X 0,Y 573.008,Z 340.194,A -85,B 0,C 180,E1 -2022.972,E2 -2022.972} C_VEL
LIN {X 0,Y 572.965,Z 342.294,A -85,B 0,C 180,E1 -2023.641,E2 -2023.641} C_VEL
LIN {X 0,Y 572.972,Z 344.676,A -85,B 0,C 180,E1 -2024.65,E2 -2024.65} C_VEL
LIN {X 0,Y 572.955,Z 346.187,A -85,B 0,C 180,E1 -2025.64,E2 -2025.64} C_VEL
LIN {X 0,Y 572.922,Z 346.909,A -85,B 0,C 180,E1 -2026.612,E2 -2026.612} C_VEL
LIN {X 0,Y 572.972,Z 346.885,A -85,B 0,C 180,E1 -2027.576,E2 -2027.576} C_VEL
LIN {X 0,Y 572.954,Z 346.107,A -85,B 0,C 180,E1 -2028.519,E2 -2028.519} C_VEL
LIN {X 0,Y 572.957,Z 343.6,A -85,B 0,C 180,E1 -2029.942,E2 -2029.942} C_VEL
LIN {X 0,Y 572.981,Z 339.632,A -85,B 0,C 180,E1 -2031.278,E2 -2031.278} C_VEL
LIN {X 0,Y 573.023,Z 334.346,A -85,B 0,C 180,E1 -2032.544,E2 -2032.544} C_VEL
LIN {X 0,Y 573.096,Z 327.816,A -85,B 0,C 180,E1 -2033.723,E2 -2033.723} C_VEL
LIN {X 0,Y 573.115,Z 320.265,A -85,B 0,C 180,E1 -2034.806,E2 -2034.806} C_VEL
LIN {X 0,Y 573.279,Z 311.897,A -85,B 0,C 180,E1 -2035.779,E2 -2035.779} C_VEL
LIN {X 0,Y 573.344,Z 302.966,A -85,B 0,C 180,E1 -2036.629,E2 -2036.629} C_VEL
LIN {X 0,Y 573.448,Z 291.963,A -85,B 0,C 180,E1 -2037.476,E2 -2037.476} C_VEL
LIN {X 0,Y 573.569,Z 281.453,A -85,B 0,C 180,E1 -2038.125,E2 -2038.125} C_VEL
LIN {X 0,Y 573.662,Z 270.237,A -85,B 0,C 180,E1 -2038.675,E2 -2038.675} C_VEL
LIN {X 0,Y 573.799,Z 257.144,A -85,B 0,C 180,E1 -2039.148,E2 -2039.148} C_VEL
LIN {X 0,Y 573.619,Z 247.929,A -85,B 0,C 180,E1 -2039.395,E2 -2039.395} C_VEL
LIN {X 0,Y 572.949,Z 243.679,A -85,B 0,C 180,E1 -2039.502,E2 -2039.502} C_VEL
LIN {X 0,Y 572.947,Z 240.073,A -85,B 0,C 180,E1 -2042.218,E2 -2042.218} C_VEL
LIN {X 0,Y 572.993,Z 236.194,A -85,B 0,C 180,E1 -2045.177,E2 -2045.177} C_VEL
LIN {X 0,Y 572.96,Z 233.016,A -85,B 0,C 180,E1 -2047.651,E2 -2047.651} C_VEL
LIN {X 0,Y 572.984,Z 230.437,A -85,B 0,C 180,E1 -2049.914,E2 -2049.914} C_VEL
LIN {X 0,Y 573.019,Z 227.895,A -85,B 0,C 180,E1 -2052.145,E2 -2052.145} C_VEL
LIN {X 0,Y 573.038,Z 225.213,A -85,B 0,C 180,E1 -2054.347,E2 -2054.347} C_VEL
LIN {X 0,Y 573.046,Z 222.699,A -85,B 0,C 180,E1 -2056.525,E2 -2056.525} C_VEL
LIN {X 0,Y 573.085,Z 219.262,A -85,B 0,C 180,E1 -2059.4,E2 -2059.4} C_VEL
LIN {X 0,Y 573.093,Z 217.583,A -85,B 0,C 180,E1 -2060.827,E2 -2060.827} C_VEL
LIN {X 0,Y 573.135,Z 217.097,A -85,B 0,C 180,E1 -2061.539,E2 -2061.539} C_VEL
LIN {X 0,Y 573.23,Z 217.084,A -85,B 0,C 180,E1 -2063.665,E2 -2063.665} C_VEL
LIN {X 0,Y 573.226,Z 217.085,A -85,B 0,C 180,E1 -2065.782,E2 -2065.782} C_VEL
LIN {X 0,Y 573.297,Z 217.074,A -85,B 0,C 180,E1 -2067.893,E2 -2067.893} C_VEL
LIN {X 0,Y 573.328,Z 217.073,A -85,B 0,C 180,E1 -2070.703,E2 -2070.703} C_VEL
LIN {X 0,Y 573.228,Z 217.082,A -85,B 0,C 180,E1 -2073.515,E2 -2073.515} C_VEL
LIN {X 0,Y 573.284,Z 217.076,A -85,B 0,C 180,E1 -2075.629,E2 -2075.629} C_VEL
LIN {X 0,Y 573.293,Z 217.074,A -85,B 0,C 180,E1 -2078.46,E2 -2078.46} C_VEL
LIN {X 0,Y 573.283,Z 217.079,A -85,B 0,C 180,E1 -2081.312,E2 -2081.312} C_VEL
LIN {X 0,Y 573.266,Z 217.077,A -85,B 0,C 180,E1 -2084.426,E2 -2084.426} C_VEL
LIN {X 0,Y 573.248,Z 217.081,A -85,B 0,C 180,E1 -2087.112,E2 -2087.112} C_VEL
LIN {X 0,Y 573.245,Z 217.08,A -85,B 0,C 180,E1 -2090.077,E2 -2090.077} C_VEL
LIN {X 0,Y 573.258,Z 217.081,A -85,B 0,C 180,E1 -2093.155,E2 -2093.155} C_VEL
LIN {X 0,Y 573.28,Z 217.076,A -85,B 0,C 180,E1 -2096.189,E2 -2096.189} C_VEL
LIN {X 0,Y 573.231,Z 217.082,A -85,B 0,C 180,E1 -2098.565,E2 -2098.565} C_VEL
LIN {X 0,Y 573.224,Z 217.083,A -85,B 0,C 180,E1 -2100.994,E2 -2100.994} C_VEL
LIN {X 0,Y 573.276,Z 217.076,A -85,B 0,C 180,E1 -2103.529,E2 -2103.529} C_VEL
LIN {X 0,Y 573.247,Z 217.08,A -85,B 0,C 180,E1 -2106.049,E2 -2106.049} C_VEL
LIN {X 0,Y 573.24,Z 217.084,A -85,B 0,C 180,E1 -2108.702,E2 -2108.702} C_VEL
LIN {X 0,Y 573.255,Z 217.079,A -85,B 0,C 180,E1 -2111.598,E2 -2111.598} C_VEL
LIN {X 0,Y 573.229,Z 217.082,A -85,B 0,C 180,E1 -2114.334,E2 -2114.334} C_VEL
LIN {X 0,Y 573.235,Z 217.082,A -85,B 0,C 180,E1 -2117.359,E2 -2117.359} C_VEL
LIN {X 0,Y 573.243,Z 217.081,A -85,B 0,C 180,E1 -2120.395,E2 -2120.395} C_VEL
LIN {X 0,Y 573.25,Z 217.082,A -85,B 0,C 180,E1 -2123.079,E2 -2123.079} C_VEL
LIN {X 0,Y 573.265,Z 217.079,A -85,B 0,C 180,E1 -2125.673,E2 -2125.673} C_VEL
LIN {X 0,Y 573.244,Z 217.081,A -85,B 0,C 180,E1 -2128.187,E2 -2128.187} C_VEL
LIN {X 0,Y 573.265,Z 217.078,A -85,B 0,C 180,E1 -2130.636,E2 -2130.636} C_VEL
LIN {X 0,Y 573.246,Z 217.08,A -85,B 0,C 180,E1 -2133.026,E2 -2133.026} C_VEL
LIN {X 0,Y 573.272,Z 217.077,A -85,B 0,C 180,E1 -2135.368,E2 -2135.368} C_VEL
LIN {X 0,Y 573.228,Z 217.085,A -85,B 0,C 180,E1 -2138.421,E2 -2138.421} C_VEL
LIN {X 0,Y 573.276,Z 217.078,A -85,B 0,C 180,E1 -2140.73,E2 -2140.73} C_VEL
LIN {X 0,Y 573.258,Z 217.08,A -85,B 0,C 180,E1 -2143.623,E2 -2143.623} C_VEL
LIN {X 0,Y 573.271,Z 217.08,A -85,B 0,C 180,E1 -2145.808,E2 -2145.808} C_VEL
LIN {X 0,Y 573.263,Z 217.078,A -85,B 0,C 180,E1 -2148.746,E2 -2148.746} C_VEL
LIN {X 0,Y 573.245,Z 217.082,A -85,B 0,C 180,E1 -2151.541,E2 -2151.541} C_VEL
LIN {X 0,Y 573.252,Z 217.08,A -85,B 0,C 180,E1 -2153.666,E2 -2153.666} C_VEL
LIN {X 0,Y 573.228,Z 217.082,A -85,B 0,C 180,E1 -2155.783,E2 -2155.783} C_VEL
LIN {X 0,Y 573.301,Z 217.074,A -85,B 0,C 180,E1 -2157.894,E2 -2157.894} C_VEL
LIN {X 0,Y 573.327,Z 217.07,A -85,B 0,C 180,E1 -2160.704,E2 -2160.704} C_VEL
LIN {X 0,Y 573.232,Z 217.084,A -85,B 0,C 180,E1 -2163.516,E2 -2163.516} C_VEL
LIN {X 0,Y 573.293,Z 217.075,A -85,B 0,C 180,E1 -2165.629,E2 -2165.629} C_VEL
LIN {X 0,Y 573.258,Z 217.081,A -85,B 0,C 180,E1 -2168.461,E2 -2168.461} C_VEL
LIN {X 0,Y 573.277,Z 217.076,A -85,B 0,C 180,E1 -2171.313,E2 -2171.313} C_VEL
LIN {X 0,Y 573.281,Z 217.078,A -85,B 0,C 180,E1 -2174.423,E2 -2174.423} C_VEL
LIN {X 0,Y 573.265,Z 217.078,A -85,B 0,C 180,E1 -2177.112,E2 -2177.112} C_VEL
LIN {X 0,Y 573.246,Z 217.082,A -85,B 0,C 180,E1 -2180.078,E2 -2180.078} C_VEL
LIN {X 0,Y 573.239,Z 217.081,A -85,B 0,C 180,E1 -2182.339,E2 -2182.339} C_VEL
LIN {X 0,Y 573.241,Z 217.081,A -85,B 0,C 180,E1 -2185.412,E2 -2185.412} C_VEL
LIN {X 0,Y 573.256,Z 217.078,A -85,B 0,C 180,E1 -2188.029,E2 -2188.029} C_VEL
LIN {X 0,Y 573.241,Z 217.081,A -85,B 0,C 180,E1 -2190.177,E2 -2190.177} C_VEL
LIN {X 0,Y 573.258,Z 217.079,A -85,B 0,C 180,E1 -2192.646,E2 -2192.646} C_VEL
LIN {X 0,Y 573.214,Z 217.084,A -85,B 0,C 180,E1 -2195.188,E2 -2195.188} C_VEL
LIN {X 0,Y 573.241,Z 217.081,A -85,B 0,C 180,E1 -2197.808,E2 -2197.808} C_VEL
LIN {X 0,Y 573.25,Z 217.083,A -85,B 0,C 180,E1 -2200.525,E2 -2200.525} C_VEL
LIN {X 0,Y 573.243,Z 217.08,A -85,B 0,C 180,E1 -2203.359,E2 -2203.359} C_VEL
LIN {X 0,Y 573.244,Z 217.082,A -85,B 0,C 180,E1 -2206.332,E2 -2206.332} C_VEL
LIN {X 0,Y 573.235,Z 217.082,A -85,B 0,C 180,E1 -2208.543,E2 -2208.543} C_VEL
LIN {X 0,Y 573.249,Z 217.083,A -85,B 0,C 180,E1 -2211.299,E2 -2211.299} C_VEL
LIN {X 0,Y 573.293,Z 217.284,A -85,B 0,C 180,E1 -2213.3,E2 -2213.3} C_VEL
LIN {X 0,Y 573.79,Z 221.916,A -85,B 0,C 180,E1 -2214.853,E2 -2214.853} C_VEL
LIN {X 0,Y 573.664,Z 229.859,A -85,B 0,C 180,E1 -2217.381,E2 -2217.381} C_VEL
LIN {X 0,Y 573.613,Z 238.938,A -85,B 0,C 180,E1 -2220.192,E2 -2220.192} C_VEL
LIN {X 0,Y 573.458,Z 248.394,A -85,B 0,C 180,E1 -2223.034,E2 -2223.034} C_VEL
LIN {X 0,Y 573.395,Z 257.661,A -85,B 0,C 180,E1 -2225.757,E2 -2225.757} C_VEL
LIN {X 0,Y 573.325,Z 266.928,A -85,B 0,C 180,E1 -2228.423,E2 -2228.423} C_VEL
LIN {X 0,Y 573.222,Z 276.329,A -85,B 0,C 180,E1 -2231.077,E2 -2231.077} C_VEL
LIN {X 0,Y 573.164,Z 286.786,A -85,B 0,C 180,E1 -2233.985,E2 -2233.985} C_VEL
LIN {X 0,Y 573.097,Z 297.378,A -85,B 0,C 180,E1 -2236.887,E2 -2236.887} C_VEL
LIN {X 0,Y 573.083,Z 299.529,A -85,B 0,C 180,E1 -2237.472,E2 -2237.472} C_VEL
LIN {X 0,Y 573.867,Z 306.354,A -85,B 0,C 180,E1 -2237.624,E2 -2237.624} C_VEL
LIN {X 0,Y 573.78,Z 318.485,A -85,B 0,C 180,E1 -2237.936,E2 -2237.936} C_VEL
LIN {X 0,Y 573.644,Z 330.519,A -85,B 0,C 180,E1 -2238.382,E2 -2238.382} C_VEL
LIN {X 0,Y 573.512,Z 342.472,A -85,B 0,C 180,E1 -2238.976,E2 -2238.976} C_VEL
LIN {X 0,Y 573.455,Z 353.473,A -85,B 0,C 180,E1 -2239.674,E2 -2239.674} C_VEL
LIN {X 0,Y 573.308,Z 363.643,A -85,B 0,C 180,E1 -2240.474,E2 -2240.474} C_VEL
LIN {X 0,Y 573.207,Z 372.784,A -85,B 0,C 180,E1 -2241.361,E2 -2241.361} C_VEL
LIN {X 0,Y 573.143,Z 381.688,A -85,B 0,C 180,E1 -2242.425,E2 -2242.425} C_VEL
LIN {X 0,Y 573.051,Z 388.407,A -85,B 0,C 180,E1 -2243.415,E2 -2243.415} C_VEL
LIN {X 0,Y 573.071,Z 393.678,A -85,B 0,C 180,E1 -2244.369,E2 -2244.369} C_VEL
LIN {X 0,Y 573.029,Z 398.37,A -85,B 0,C 180,E1 -2245.427,E2 -2245.427} C_VEL
LIN {X 0,Y 573.022,Z 401.955,A -85,B 0,C 180,E1 -2246.484,E2 -2246.484} C_VEL
LIN {X 0,Y 572.959,Z 403.808,A -85,B 0,C 180,E1 -2247.187,E2 -2247.187} C_VEL
LIN {X 0,Y 572.94,Z 405.2,A -85,B 0,C 180,E1 -2247.891,E2 -2247.891} C_VEL
LIN {X 0,Y 572.94,Z 406.784,A -85,B 0,C 180,E1 -2249.297,E2 -2249.297} C_VEL
LIN {X 0,Y 572.938,Z 407,A -85,B 0,C 180,E1 -2250,E2 -2250} C_VEL
LIN {X 0,Y 572.946,Z 406.185,A -85,B 0,C 180,E1 -2251.405,E2 -2251.405} C_VEL
LIN {X 0,Y 572.94,Z 405.202,A -85,B 0,C 180,E1 -2252.109,E2 -2252.109} C_VEL
LIN {X 0,Y 572.959,Z 403.811,A -85,B 0,C 180,E1 -2252.812,E2 -2252.812} C_VEL
LIN {X 0,Y 573.015,Z 400.897,A -85,B 0,C 180,E1 -2253.868,E2 -2253.868} C_VEL
LIN {X 0,Y 572.963,Z 396.951,A -85,B 0,C 180,E1 -2254.925,E2 -2254.925} C_VEL
LIN {X 0,Y 573.065,Z 390.88,A -85,B 0,C 180,E1 -2256.16,E2 -2256.16} C_VEL
LIN {X 0,Y 573.12,Z 384.239,A -85,B 0,C 180,E1 -2257.22,E2 -2257.22} C_VEL
LIN {X 0,Y 573.201,Z 375.993,A -85,B 0,C 180,E1 -2258.283,E2 -2258.283} C_VEL
LIN {X 0,Y 573.287,Z 367.542,A -85,B 0,C 180,E1 -2259.17,E2 -2259.17} C_VEL
LIN {X 0,Y 573.43,Z 357.1,A -85,B 0,C 180,E1 -2260.058,E2 -2260.058} C_VEL
LIN {X 0,Y 573.512,Z 345.542,A -85,B 0,C 180,E1 -2260.847,E2 -2260.847} C_VEL
LIN {X 0,Y 573.611,Z 333.889,A -85,B 0,C 180,E1 -2261.466,E2 -2261.466} C_VEL
LIN {X 0,Y 573.733,Z 321.188,A -85,B 0,C 180,E1 -2261.974,E2 -2261.974} C_VEL
LIN {X 0,Y 573.866,Z 308.54,A -85,B 0,C 180,E1 -2262.33,E2 -2262.33} C_VEL
LIN {X 0,Y 573.573,Z 302.674,A -85,B 0,C 180,E1 -2262.455,E2 -2262.455} C_VEL
LIN {X 0,Y 573.083,Z 299.532,A -85,B 0,C 180,E1 -2262.527,E2 -2262.527} C_VEL
LIN {X 0,Y 573.158,Z 289.437,A -85,B 0,C 180,E1 -2265.285,E2 -2265.285} C_VEL
LIN {X 0,Y 573.215,Z 278.846,A -85,B 0,C 180,E1 -2268.218,E2 -2268.218} C_VEL
LIN {X 0,Y 573.301,Z 269.579,A -85,B 0,C 180,E1 -2270.824,E2 -2270.824} C_VEL
LIN {X 0,Y 573.369,Z 260.313,A -85,B 0,C 180,E1 -2273.475,E2 -2273.475} C_VEL
LIN {X 0,Y 573.453,Z 251.044,A -85,B 0,C 180,E1 -2276.18,E2 -2276.18} C_VEL
LIN {X 0,Y 573.506,Z 241.777,A -85,B 0,C 180,E1 -2278.95,E2 -2278.95} C_VEL
LIN {X 0,Y 573.627,Z 233.834,A -85,B 0,C 180,E1 -2281.379,E2 -2281.379} C_VEL
LIN {X 0,Y 573.774,Z 224.566,A -85,B 0,C 180,E1 -2284.293,E2 -2284.293} C_VEL
LIN {X 0,Y 573.623,Z 219.222,A -85,B 0,C 180,E1 -2286.037,E2 -2286.037} C_VEL
LIN {X 0,Y 573.262,Z 217.081,A -85,B 0,C 180,E1 -2286.811,E2 -2286.811} C_VEL
LIN {X 0,Y 573.238,Z 217.083,A -85,B 0,C 180,E1 -2289.607,E2 -2289.607} C_VEL
LIN {X 0,Y 573.242,Z 217.083,A -85,B 0,C 180,E1 -2292.641,E2 -2292.641} C_VEL
LIN {X 0,Y 573.236,Z 217.084,A -85,B 0,C 180,E1 -2295.666,E2 -2295.666} C_VEL
LIN {X 0,Y 573.246,Z 217.083,A -85,B 0,C 180,E1 -2298.544,E2 -2298.544} C_VEL
LIN {X 0,Y 573.25,Z 217.08,A -85,B 0,C 180,E1 -2301.298,E2 -2301.298} C_VEL
LIN {X 0,Y 573.213,Z 217.087,A -85,B 0,C 180,E1 -2304.017,E2 -2304.017} C_VEL
LIN {X 0,Y 573.269,Z 217.078,A -85,B 0,C 180,E1 -2306.517,E2 -2306.517} C_VEL
LIN {X 0,Y 573.233,Z 217.085,A -85,B 0,C 180,E1 -2309.116,E2 -2309.116} C_VEL
LIN {X 0,Y 573.252,Z 217.081,A -85,B 0,C 180,E1 -2311.97,E2 -2311.97} C_VEL
LIN {X 0,Y 573.257,Z 217.08,A -85,B 0,C 180,E1 -2314.589,E2 -2314.589} C_VEL
LIN {X 0,Y 573.237,Z 217.082,A -85,B 0,C 180,E1 -2317.661,E2 -2317.661} C_VEL
LIN {X 0,Y 573.255,Z 217.079,A -85,B 0,C 180,E1 -2319.923,E2 -2319.923} C_VEL
